SPLINE
SPL {X  -141.034, Y  +747.040, Z    +0.000, E1  +398.619, E3 -227248.265}
SPL {X  -152.334, Y  +720.400, Z    +0.000, E1  +389.143, E3 -227267.719}
SPL {X  -157.190, Y  +701.303, Z    +0.000, E1  +380.164, E3 -227274.880}
SPL {X  -159.117, Y  +688.191, Z    +0.000, E1  +372.748, E3 -227277.912}
SPL {X  -159.875, Y  +677.561, Z    +0.000, E1  +366.083, E3 -227279.302}
SPL {X  -159.990, Y  +669.975, Z    +0.000, E1  +360.595, E3 -227279.733}
SPL {X  -159.990, Y  +666.850, Z    +0.000, E1  +357.321, E3 -227279.833}
SPL {X  -159.990, Y  +662.495, Z    +0.000, E1  +351.318, E3 -227280.128}
SPL {X  -159.990, Y  +657.714, Z    +0.000, E1  +344.114, E3 -227280.689}
SPL {X  -159.990, Y  +651.822, Z    +0.000, E1  +335.261, E3 -227281.657}
SPL {X  -159.990, Y  +641.369, Z    +0.000, E1  +322.665, E3 -227284.495}
SPL {X  -159.990, Y  +598.251, Z    +0.000, E1  +304.104, E3 -227308.266}
SPL {X  -159.990, Y  +514.954, Z    +0.000, E1  +299.688, E3 -227382.062}
SPL {X  -159.990, Y  +505.641, Z    +0.000, E1  +299.707, E3 -227393.371}
SPL {X  -159.990, Y  +498.210, Z    +0.000, E1  +299.707, E3 -227402.364}
SPL {X  -159.990, Y  +488.988, Z    +0.000, E1  +299.693, E3 -227413.501}
SPL {X  -159.990, Y  +478.987, Z    +0.000, E1  +299.694, E3 -227425.604}
SPL {X  -159.990, Y  +468.796, Z    +0.000, E1  +299.698, E3 -227437.948}
SPL {X  -159.990, Y  +460.399, Z    +0.000, E1  +299.707, E3 -227448.124}
SPL {X  -159.990, Y  +453.289, Z    +0.000, E1  +299.707, E3 -227456.730}
SPL {X  -159.990, Y  +443.890, Z    +0.000, E1  +299.691, E3 -227468.083}
SPL {X  -159.990, Y  +437.910, Z    +0.000, E1  +300.175, E3 -227478.554}
ENDSPLINE

SPLINE
SPL {X  -159.990, Y  +447.165, Z    +0.000, E1  +303.287, E3 -227487.109}
ENDSPLINE

SPLINE
SPL {X  -159.990, Y  +436.354, Z    +0.000, E1  +302.683, E3 -227498.121}
SPL {X  -159.990, Y  +425.140, Z    +0.000, E1  +301.982, E3 -227508.556}
SPL {X  -159.990, Y  +412.625, Z    +0.000, E1  +301.150, E3 -227519.392}
SPL {X  -159.990, Y  +398.951, Z    +0.000, E1  +300.353, E3 -227531.264}
SPL {X  -159.990, Y  +389.564, Z    +0.000, E1  +300.093, E3 -227541.078}
SPL {X  -159.985, Y  +381.230, Z    +0.000, E1  +300.090, E3 -227551.345}
SPL {X  -159.702, Y  +372.900, Z    +0.000, E1  +300.135, E3 -227561.882}
SPL {X  -159.030, Y  +365.001, Z    +0.000, E1  +300.230, E3 -227572.284}
SPL {X  -157.449, Y  +354.098, Z    +0.000, E1  +300.447, E3 -227587.284}
SPL {X  -155.503, Y  +344.875, Z    +0.000, E1  +300.798, E3 -227600.703}
SPL {X  -153.622, Y  +337.813, Z    +0.000, E1  +301.097, E3 -227611.296}
SPL {X  -150.877, Y  +329.275, Z    +0.000, E1  +301.527, E3 -227624.521}
SPL {X  -148.134, Y  +322.059, Z    +0.000, E1  +302.038, E3 -227636.159}
SPL {X  -145.832, Y  +316.699, Z    +0.000, E1  +302.442, E3 -227644.994}
SPL {X  -143.160, Y  +311.071, Z    +0.000, E1  +302.918, E3 -227654.439}
SPL {X  -140.427, Y  +305.839, Z    +0.000, E1  +303.430, E3 -227663.400}
SPL {X  -137.611, Y  +300.891, Z    +0.000, E1  +303.950, E3 -227671.976}
SPL {X  -121.335, Y  +278.219, Z    +0.000, E1  +311.699, E3 -227770.322}
ENDSPLINE

SPLINE
SPL {X  -146.770, Y  +318.818, Z    +0.000, E1  +325.496, E3 -227870.156}
SPL {X  -156.430, Y  +348.936, Z    +0.000, E1  +338.153, E3 -227886.887}
SPL {X  -159.088, Y  +365.539, Z    +0.000, E1  +347.196, E3 -227891.298}
SPL {X  -159.820, Y  +375.127, Z    +0.000, E1  +353.170, E3 -227892.722}
SPL {X  -159.990, Y  +382.134, Z    +0.000, E1  +357.935, E3 -227893.240}
SPL {X  -159.990, Y  +385.595, Z    +0.000, E1  +360.838, E3 -227893.355}
SPL {X  -159.990, Y  +390.176, Z    +0.000, E1  +366.367, E3 -227893.624}
SPL {X  -159.990, Y  +395.747, Z    +0.000, E1  +374.484, E3 -227894.250}
SPL {X  -159.990, Y  +404.190, Z    +0.000, E1  +386.444, E3 -227895.932}
SPL {X  -159.990, Y  +418.143, Z    +0.000, E1  +401.167, E3 -227900.525}
SPL {X  -159.990, Y  +460.468, Z    +0.000, E1  +416.751, E3 -227923.207}
SPL {X  -159.990, Y  +537.348, Z    +0.000, E1  +420.157, E3 -227993.218}
SPL {X  -159.990, Y  +545.972, Z    +0.000, E1  +420.143, E3 -228003.752}
SPL {X  -159.990, Y  +557.131, Z    +0.000, E1  +420.184, E3 -228017.266}
SPL {X  -159.990, Y  +569.073, Z    +0.000, E1  +420.153, E3 -228031.861}
SPL {X  -159.990, Y  +577.562, Z    +0.000, E1  +420.146, E3 -228042.201}
SPL {X  -159.990, Y  +585.415, Z    +0.000, E1  +420.147, E3 -228051.767}
SPL {X  -159.990, Y  +594.125, Z    +0.000, E1  +420.153, E3 -228062.353}
SPL {X  -159.990, Y  +602.716, Z    +0.000, E1  +420.150, E3 -228072.816}
SPL {X  -159.990, Y  +612.205, Z    +0.000, E1  +420.159, E3 -228084.352}
SPL {X  -159.990, Y  +620.604, Z    +0.000, E1  +420.153, E3 -228094.568}
SPL {X  -159.990, Y  +632.106, Z    +0.000, E1  +420.183, E3 -228108.544}
SPL {X  -159.990, Y  +643.341, Z    +0.000, E1  +420.148, E3 -228122.288}
SPL {X  -159.990, Y  +652.098, Z    +0.000, E1  +420.153, E3 -228132.933}
SPL {X  -159.990, Y  +661.466, Z    +0.000, E1  +420.154, E3 -228144.345}
SPL {X  -159.990, Y  +670.781, Z    +0.000, E1  +420.150, E3 -228155.692}
SPL {X  -159.839, Y  +678.445, Z    +0.000, E1  +420.123, E3 -228165.172}
SPL {X  -159.339, Y  +685.922, Z    +0.000, E1  +420.057, E3 -228174.774}
SPL {X  -158.381, Y  +694.132, Z    +0.000, E1  +419.909, E3 -228185.771}
SPL {X  -157.192, Y  +701.291, Z    +0.000, E1  +419.715, E3 -228195.742}
SPL {X  -155.426, Y  +709.440, Z    +0.000, E1  +419.459, E3 -228207.440}
SPL {X  -153.239, Y  +717.485, Z    +0.000, E1  +419.087, E3 -228219.485}
SPL {X  -151.467, Y  +723.022, Z    +0.000, E1  +418.780, E3 -228228.037}
SPL {X  -148.791, Y  +730.306, Z    +0.000, E1  +418.370, E3 -228239.502}
SPL {X  -145.943, Y  +737.055, Z    +0.000, E1  +417.829, E3 -228250.555}
SPL {X  -143.898, Y  +741.430, Z    +0.000, E1  +417.467, E3 -228257.825}
SPL {X  -141.624, Y  +745.927, Z    +0.000, E1  +417.045, E3 -228265.420}
SPL {X  -139.581, Y  +749.692, Z    +0.000, E1  +416.662, E3 -228271.866}
SPL {X  -137.120, Y  +753.931, Z    +0.000, E1  +416.213, E3 -228279.164}
SPL {X  -120.054, Y  +777.254, Z    +0.000, E1  +409.463, E3 -228365.910}
ENDSPLINE

SPLINE
SPL {X  -141.034, Y  +747.040, Z    +0.000, E1  +398.619, E3 -228474.072}
SPL {X  -152.334, Y  +720.400, Z    +0.000, E1  +389.143, E3 -228493.526}
SPL {X  -157.190, Y  +701.303, Z    +0.000, E1  +380.164, E3 -228500.687}
SPL {X  -159.117, Y  +688.191, Z    +0.000, E1  +372.748, E3 -228503.719}
SPL {X  -159.875, Y  +677.561, Z    +0.000, E1  +366.083, E3 -228505.108}
SPL {X  -159.990, Y  +671.043, Z    +0.000, E1  +361.371, E3 -228505.512}
SPL {X  -159.990, Y  +668.657, Z    +0.000, E1  +359.332, E3 -228505.573}
SPL {X  -159.990, Y  +665.812, Z    +0.000, E1  +355.875, E3 -228505.684}
SPL {X  -159.990, Y  +662.495, Z    +0.000, E1  +351.318, E3 -228505.934}
SPL {X  -159.990, Y  +657.714, Z    +0.000, E1  +344.114, E3 -228506.495}
SPL {X  -159.990, Y  +651.822, Z    +0.000, E1  +335.261, E3 -228507.463}
SPL {X  -159.990, Y  +641.369, Z    +0.000, E1  +322.665, E3 -228510.301}
SPL {X  -159.990, Y  +598.251, Z    +0.000, E1  +304.104, E3 -228534.073}
SPL {X  -159.990, Y  +514.954, Z    +0.000, E1  +299.688, E3 -228607.868}
SPL {X  -159.990, Y  +505.641, Z    +0.000, E1  +299.707, E3 -228619.177}
SPL {X  -159.990, Y  +498.210, Z    +0.000, E1  +299.707, E3 -228628.171}
SPL {X  -159.990, Y  +488.988, Z    +0.000, E1  +299.693, E3 -228639.308}
SPL {X  -159.990, Y  +478.987, Z    +0.000, E1  +299.694, E3 -228651.410}
SPL {X  -159.990, Y  +468.796, Z    +0.000, E1  +299.698, E3 -228663.754}
SPL {X  -159.990, Y  +456.606, Z    +0.000, E1  +299.670, E3 -228678.460}
SPL {X  -159.990, Y  +443.890, Z    +0.000, E1  +299.691, E3 -228693.890}
SPL {X  -159.990, Y  +437.910, Z    +0.000, E1  +300.175, E3 -228704.361}
ENDSPLINE

SPLINE
SPL {X  -159.990, Y  +447.165, Z    +0.000, E1  +303.287, E3 -228712.916}
ENDSPLINE

SPLINE
SPL {X  -159.990, Y  +436.354, Z    +0.000, E1  +302.683, E3 -228723.927}
SPL {X  -159.990, Y  +425.140, Z    +0.000, E1  +301.982, E3 -228734.363}
SPL {X  -159.990, Y  +412.625, Z    +0.000, E1  +301.150, E3 -228745.199}
SPL {X  -159.990, Y  +398.951, Z    +0.000, E1  +300.353, E3 -228757.070}
SPL {X  -159.990, Y  +389.564, Z    +0.000, E1  +300.093, E3 -228766.884}
SPL {X  -159.985, Y  +381.230, Z    +0.000, E1  +300.090, E3 -228777.151}
SPL {X  -159.702, Y  +372.900, Z    +0.000, E1  +300.135, E3 -228787.688}
SPL {X  -159.030, Y  +365.001, Z    +0.000, E1  +300.230, E3 -228798.091}
SPL {X  -157.449, Y  +354.098, Z    +0.000, E1  +300.447, E3 -228813.090}
SPL {X  -155.503, Y  +344.875, Z    +0.000, E1  +300.798, E3 -228826.509}
SPL {X  -153.622, Y  +337.813, Z    +0.000, E1  +301.097, E3 -228837.102}
SPL {X  -151.786, Y  +331.925, Z    +0.000, E1  +301.419, E3 -228846.223}
SPL {X  -150.141, Y  +327.233, Z    +0.000, E1  +301.695, E3 -228853.632}
SPL {X  -148.134, Y  +322.059, Z    +0.000, E1  +302.038, E3 -228861.966}
SPL {X  -145.832, Y  +316.699, Z    +0.000, E1  +302.442, E3 -228870.800}
SPL {X  -143.160, Y  +311.071, Z    +0.000, E1  +302.918, E3 -228880.245}
SPL {X  -140.427, Y  +305.839, Z    +0.000, E1  +303.430, E3 -228889.207}
SPL {X  -137.611, Y  +300.891, Z    +0.000, E1  +303.950, E3 -228897.783}
SPL {X  -121.335, Y  +278.219, Z    +0.000, E1  +311.699, E3 -228996.129}
ENDSPLINE

SPLINE
SPL {X  -146.770, Y  +318.818, Z    +0.000, E1  +325.496, E3 -229095.963}
SPL {X  -156.430, Y  +348.936, Z    +0.000, E1  +338.153, E3 -229112.694}
SPL {X  -159.088, Y  +365.539, Z    +0.000, E1  +347.196, E3 -229117.105}
SPL {X  -159.921, Y  +377.798, Z    +0.000, E1  +354.872, E3 -229118.765}
SPL {X  -159.990, Y  +384.169, Z    +0.000, E1  +359.534, E3 -229119.120}
SPL {X  -159.990, Y  +386.366, Z    +0.000, E1  +361.774, E3 -229119.185}
SPL {X  -159.990, Y  +390.176, Z    +0.000, E1  +366.367, E3 -229119.431}
SPL {X  -159.990, Y  +395.747, Z    +0.000, E1  +374.484, E3 -229120.056}
SPL {X  -159.990, Y  +402.387, Z    +0.000, E1  +384.140, E3 -229121.289}
SPL {X  -159.990, Y  +414.244, Z    +0.000, E1  +397.704, E3 -229124.921}
SPL {X  -159.990, Y  +460.468, Z    +0.000, E1  +416.751, E3 -229149.013}
SPL {X  -159.990, Y  +537.348, Z    +0.000, E1  +420.157, E3 -229219.025}
SPL {X  -159.990, Y  +549.907, Z    +0.000, E1  +420.183, E3 -229234.282}
SPL {X  -159.990, Y  +560.677, Z    +0.000, E1  +420.145, E3 -229247.453}
SPL {X  -159.990, Y  +569.073, Z    +0.000, E1  +420.153, E3 -229257.668}
SPL {X  -159.990, Y  +577.562, Z    +0.000, E1  +420.146, E3 -229268.008}
SPL {X  -159.990, Y  +585.415, Z    +0.000, E1  +420.147, E3 -229277.573}
SPL {X  -159.990, Y  +594.125, Z    +0.000, E1  +420.153, E3 -229288.159}
SPL {X  -159.990, Y  +602.716, Z    +0.000, E1  +420.150, E3 -229298.622}
SPL {X  -159.990, Y  +612.205, Z    +0.000, E1  +420.159, E3 -229310.159}
SPL {X  -159.990, Y  +624.752, Z    +0.000, E1  +420.194, E3 -229325.367}
SPL {X  -159.990, Y  +640.062, Z    +0.000, E1  +420.188, E3 -229344.030}
SPL {X  -159.990, Y  +652.098, Z    +0.000, E1  +420.153, E3 -229358.740}
SPL {X  -159.990, Y  +661.466, Z    +0.000, E1  +420.154, E3 -229370.151}
SPL {X  -159.963, Y  +674.441, Z    +0.000, E1  +420.189, E3 -229385.902}
SPL {X  -159.339, Y  +685.922, Z    +0.000, E1  +420.057, E3 -229400.581}
SPL {X  -158.381, Y  +694.132, Z    +0.000, E1  +419.909, E3 -229411.578}
SPL {X  -156.712, Y  +703.719, Z    +0.000, E1  +419.674, E3 -229424.943}
SPL {X  -154.922, Y  +711.450, Z    +0.000, E1  +419.348, E3 -229436.259}
SPL {X  -153.239, Y  +717.485, Z    +0.000, E1  +419.087, E3 -229445.291}
SPL {X  -150.608, Y  +725.483, Z    +0.000, E1  +418.677, E3 -229457.637}
SPL {X  -148.008, Y  +732.249, Z    +0.000, E1  +418.192, E3 -229468.503}
SPL {X  -145.943, Y  +737.055, Z    +0.000, E1  +417.829, E3 -229476.362}
SPL {X  -143.898, Y  +741.430, Z    +0.000, E1  +417.467, E3 -229483.631}
SPL {X  -141.624, Y  +745.927, Z    +0.000, E1  +417.045, E3 -229491.226}
SPL {X  -139.581, Y  +749.692, Z    +0.000, E1  +416.662, E3 -229497.673}
SPL {X  -137.120, Y  +753.931, Z    +0.000, E1  +416.213, E3 -229504.970}
SPL {X  -120.054, Y  +777.254, Z    +0.000, E1  +409.463, E3 -229591.716}
ENDSPLINE

SPLINE
SPL {X  -141.034, Y  +747.040, Z    +0.000, E1  +398.619, E3 -229699.878}
SPL {X  -152.334, Y  +720.400, Z    +0.000, E1  +389.143, E3 -229719.332}
SPL {X  -157.190, Y  +701.303, Z    +0.000, E1  +380.164, E3 -229726.493}
SPL {X  -159.460, Y  +684.516, Z    +0.000, E1  +370.556, E3 -229730.089}
SPL {X  -159.938, Y  +675.597, Z    +0.000, E1  +364.669, E3 -229731.095}
SPL {X  -159.990, Y  +671.043, Z    +0.000, E1  +361.371, E3 -229731.319}
SPL {X  -159.990, Y  +668.657, Z    +0.000, E1  +359.332, E3 -229731.379}
SPL {X  -159.990, Y  +665.812, Z    +0.000, E1  +355.875, E3 -229731.491}
SPL {X  -159.990, Y  +662.495, Z    +0.000, E1  +351.318, E3 -229731.740}
SPL {X  -159.990, Y  +657.714, Z    +0.000, E1  +344.114, E3 -229732.302}
SPL {X  -159.990, Y  +651.822, Z    +0.000, E1  +335.261, E3 -229733.270}
SPL {X  -159.990, Y  +641.369, Z    +0.000, E1  +322.665, E3 -229736.108}
SPL {X  -159.990, Y  +598.251, Z    +0.000, E1  +304.104, E3 -229759.879}
SPL {X  -159.990, Y  +514.954, Z    +0.000, E1  +299.688, E3 -229833.675}
SPL {X  -159.990, Y  +505.641, Z    +0.000, E1  +299.707, E3 -229844.984}
SPL {X  -159.990, Y  +498.210, Z    +0.000, E1  +299.707, E3 -229853.977}
SPL {X  -159.990, Y  +488.988, Z    +0.000, E1  +299.693, E3 -229865.114}
SPL {X  -159.990, Y  +478.987, Z    +0.000, E1  +299.694, E3 -229877.217}
SPL {X  -159.990, Y  +468.796, Z    +0.000, E1  +299.698, E3 -229889.561}
SPL {X  -159.990, Y  +456.606, Z    +0.000, E1  +299.670, E3 -229904.266}
SPL {X  -159.990, Y  +443.890, Z    +0.000, E1  +299.691, E3 -229919.696}
SPL {X  -159.990, Y  +437.910, Z    +0.000, E1  +300.175, E3 -229930.167}
ENDSPLINE

SPLINE
SPL {X  -159.990, Y  +447.165, Z    +0.000, E1  +303.287, E3 -229938.722}
ENDSPLINE

SPLINE
SPL {X  -159.990, Y  +436.354, Z    +0.000, E1  +302.683, E3 -229949.734}
SPL {X  -159.990, Y  +425.140, Z    +0.000, E1  +301.982, E3 -229960.169}
SPL {X  -159.990, Y  +412.625, Z    +0.000, E1  +301.150, E3 -229971.005}
SPL {X  -159.990, Y  +398.951, Z    +0.000, E1  +300.353, E3 -229982.877}
SPL {X  -159.990, Y  +389.564, Z    +0.000, E1  +300.093, E3 -229992.690}
SPL {X  -159.985, Y  +381.230, Z    +0.000, E1  +300.090, E3 -230002.957}
SPL {X  -159.702, Y  +372.900, Z    +0.000, E1  +300.135, E3 -230013.494}
SPL {X  -159.030, Y  +365.001, Z    +0.000, E1  +300.230, E3 -230023.897}
SPL {X  -158.029, Y  +357.528, Z    +0.000, E1  +300.403, E3 -230034.153}
SPL {X  -156.953, Y  +351.476, Z    +0.000, E1  +300.570, E3 -230042.706}
SPL {X  -155.503, Y  +344.875, Z    +0.000, E1  +300.798, E3 -230052.316}
SPL {X  -153.622, Y  +337.813, Z    +0.000, E1  +301.097, E3 -230062.909}
SPL {X  -150.877, Y  +329.275, Z    +0.000, E1  +301.527, E3 -230076.134}
SPL {X  -148.134, Y  +322.059, Z    +0.000, E1  +302.038, E3 -230087.772}
SPL {X  -145.832, Y  +316.699, Z    +0.000, E1  +302.442, E3 -230096.607}
SPL {X  -143.160, Y  +311.071, Z    +0.000, E1  +302.918, E3 -230106.052}
SPL {X  -139.570, Y  +304.288, Z    +0.000, E1  +303.552, E3 -230117.648}
SPL {X  -136.734, Y  +299.430, Z    +0.000, E1  +304.147, E3 -230126.186}
SPL {X  -121.335, Y  +278.219, Z    +0.000, E1  +311.699, E3 -230221.935}
ENDSPLINE

SPLINE
SPL {X  -146.770, Y  +318.818, Z    +0.000, E1  +325.496, E3 -230321.769}
SPL {X  -156.430, Y  +348.936, Z    +0.000, E1  +338.153, E3 -230338.500}
SPL {X  -159.088, Y  +365.539, Z    +0.000, E1  +347.196, E3 -230342.911}
SPL {X  -159.921, Y  +377.798, Z    +0.000, E1  +354.872, E3 -230344.571}
SPL {X  -159.990, Y  +383.148, Z    +0.000, E1  +358.786, E3 -230344.899}
SPL {X  -159.990, Y  +384.761, Z    +0.000, E1  +360.138, E3 -230344.943}
SPL {X  -159.990, Y  +387.385, Z    +0.000, E1  +362.811, E3 -230345.045}
SPL {X  -159.990, Y  +391.439, Z    +0.000, E1  +368.259, E3 -230345.342}
SPL {X  -159.990, Y  +395.747, Z    +0.000, E1  +374.484, E3 -230345.863}
SPL {X  -159.990, Y  +402.387, Z    +0.000, E1  +384.140, E3 -230347.095}
SPL {X  -159.990, Y  +414.244, Z    +0.000, E1  +397.704, E3 -230350.728}
SPL {X  -159.990, Y  +460.468, Z    +0.000, E1  +416.751, E3 -230374.820}
SPL {X  -159.990, Y  +537.348, Z    +0.000, E1  +420.157, E3 -230444.831}
SPL {X  -159.990, Y  +549.907, Z    +0.000, E1  +420.183, E3 -230460.089}
SPL {X  -159.990, Y  +560.677, Z    +0.000, E1  +420.145, E3 -230473.260}
SPL {X  -159.990, Y  +569.073, Z    +0.000, E1  +420.153, E3 -230483.474}
SPL {X  -159.990, Y  +581.828, Z    +0.000, E1  +420.191, E3 -230498.933}
SPL {X  -159.990, Y  +594.125, Z    +0.000, E1  +420.153, E3 -230513.966}
SPL {X  -159.990, Y  +602.716, Z    +0.000, E1  +420.150, E3 -230524.429}
SPL {X  -159.990, Y  +612.205, Z    +0.000, E1  +420.159, E3 -230535.965}
SPL {X  -159.990, Y  +620.604, Z    +0.000, E1  +420.153, E3 -230546.181}
SPL {X  -159.990, Y  +632.106, Z    +0.000, E1  +420.183, E3 -230560.157}
SPL {X  -159.990, Y  +643.341, Z    +0.000, E1  +420.148, E3 -230573.901}
SPL {X  -159.990, Y  +652.098, Z    +0.000, E1  +420.153, E3 -230584.546}
SPL {X  -159.990, Y  +661.466, Z    +0.000, E1  +420.154, E3 -230595.958}
SPL {X  -159.990, Y  +670.781, Z    +0.000, E1  +420.150, E3 -230607.305}
SPL {X  -159.839, Y  +678.445, Z    +0.000, E1  +420.123, E3 -230616.785}
SPL {X  -159.339, Y  +685.922, Z    +0.000, E1  +420.057, E3 -230626.387}
SPL {X  -158.381, Y  +694.132, Z    +0.000, E1  +419.909, E3 -230637.384}
SPL {X  -157.192, Y  +701.291, Z    +0.000, E1  +419.715, E3 -230647.355}
SPL {X  -155.426, Y  +709.440, Z    +0.000, E1  +419.459, E3 -230659.053}
SPL {X  -153.239, Y  +717.485, Z    +0.000, E1  +419.087, E3 -230671.098}
SPL {X  -151.467, Y  +723.022, Z    +0.000, E1  +418.780, E3 -230679.650}
SPL {X  -148.791, Y  +730.306, Z    +0.000, E1  +418.370, E3 -230691.115}
SPL {X  -145.943, Y  +737.055, Z    +0.000, E1  +417.829, E3 -230702.168}
SPL {X  -143.898, Y  +741.430, Z    +0.000, E1  +417.467, E3 -230709.437}
SPL {X  -140.579, Y  +747.882, Z    +0.000, E1  +416.895, E3 -230720.316}
SPL {X  -137.120, Y  +753.931, Z    +0.000, E1  +416.213, E3 -230730.777}
SPL {X  -120.054, Y  +777.254, Z    +0.000, E1  +409.463, E3 -230817.523}
ENDSPLINE

SPLINE
SPL {X  -141.034, Y  +747.040, Z    +0.000, E1  +398.619, E3 -230925.685}
SPL {X  -152.334, Y  +720.400, Z    +0.000, E1  +389.143, E3 -230945.139}
SPL {X  -157.190, Y  +701.303, Z    +0.000, E1  +380.164, E3 -230952.299}
SPL {X  -159.460, Y  +684.516, Z    +0.000, E1  +370.556, E3 -230955.895}
SPL {X  -159.938, Y  +675.597, Z    +0.000, E1  +364.669, E3 -230956.902}
SPL {X  -159.990, Y  +671.043, Z    +0.000, E1  +361.371, E3 -230957.125}
SPL {X  -159.990, Y  +668.657, Z    +0.000, E1  +359.332, E3 -230957.186}
SPL {X  -159.990, Y  +665.812, Z    +0.000, E1  +355.875, E3 -230957.297}
SPL {X  -159.990, Y  +662.495, Z    +0.000, E1  +351.318, E3 -230957.547}
SPL {X  -159.990, Y  +657.714, Z    +0.000, E1  +344.114, E3 -230958.108}
SPL {X  -159.990, Y  +651.822, Z    +0.000, E1  +335.261, E3 -230959.076}
SPL {X  -159.990, Y  +641.369, Z    +0.000, E1  +322.665, E3 -230961.914}
SPL {X  -159.990, Y  +598.251, Z    +0.000, E1  +304.104, E3 -230985.686}
SPL {X  -159.990, Y  +514.954, Z    +0.000, E1  +299.688, E3 -231059.481}
SPL {X  -159.990, Y  +505.641, Z    +0.000, E1  +299.707, E3 -231070.790}
SPL {X  -159.990, Y  +498.210, Z    +0.000, E1  +299.707, E3 -231079.784}
SPL {X  -159.990, Y  +488.988, Z    +0.000, E1  +299.693, E3 -231090.921}
SPL {X  -159.990, Y  +478.987, Z    +0.000, E1  +299.694, E3 -231103.023}
SPL {X  -159.990, Y  +468.796, Z    +0.000, E1  +299.698, E3 -231115.367}
SPL {X  -159.990, Y  +460.399, Z    +0.000, E1  +299.707, E3 -231125.544}
SPL {X  -159.990, Y  +453.289, Z    +0.000, E1  +299.707, E3 -231134.149}
SPL {X  -159.990, Y  +443.890, Z    +0.000, E1  +299.691, E3 -231145.503}
SPL {X  -159.990, Y  +437.910, Z    +0.000, E1  +300.175, E3 -231155.974}
ENDSPLINE

SPLINE
SPL {X  -159.990, Y  +447.165, Z    +0.000, E1  +303.287, E3 -231164.529}
ENDSPLINE

SPLINE
SPL {X  -159.990, Y  +436.354, Z    +0.000, E1  +302.683, E3 -231175.540}
SPL {X  -159.990, Y  +425.140, Z    +0.000, E1  +301.982, E3 -231185.976}
SPL {X  -159.990, Y  +412.625, Z    +0.000, E1  +301.150, E3 -231196.812}
SPL {X  -159.990, Y  +398.951, Z    +0.000, E1  +300.353, E3 -231208.683}
SPL {X  -159.990, Y  +389.564, Z    +0.000, E1  +300.093, E3 -231218.497}
SPL {X  -159.985, Y  +381.230, Z    +0.000, E1  +300.090, E3 -231228.764}
SPL {X  -159.702, Y  +372.900, Z    +0.000, E1  +300.135, E3 -231239.301}
SPL {X  -159.030, Y  +365.001, Z    +0.000, E1  +300.230, E3 -231249.704}
SPL {X  -158.029, Y  +357.528, Z    +0.000, E1  +300.403, E3 -231259.959}
SPL {X  -156.953, Y  +351.476, Z    +0.000, E1  +300.570, E3 -231268.512}
SPL {X  -155.503, Y  +344.875, Z    +0.000, E1  +300.798, E3 -231278.122}
SPL {X  -153.622, Y  +337.813, Z    +0.000, E1  +301.097, E3 -231288.715}
SPL {X  -150.877, Y  +329.275, Z    +0.000, E1  +301.527, E3 -231301.940}
SPL {X  -148.134, Y  +322.059, Z    +0.000, E1  +302.038, E3 -231313.579}
SPL {X  -145.832, Y  +316.699, Z    +0.000, E1  +302.442, E3 -231322.413}
SPL {X  -143.160, Y  +311.071, Z    +0.000, E1  +302.918, E3 -231331.858}
SPL {X  -140.427, Y  +305.839, Z    +0.000, E1  +303.430, E3 -231340.819}
SPL {X  -137.611, Y  +300.891, Z    +0.000, E1  +303.950, E3 -231349.396}
SPL {X  -121.335, Y  +278.219, Z    +0.000, E1  +311.699, E3 -231447.742}
ENDSPLINE

SPLINE
SPL {X  -146.770, Y  +318.818, Z    +0.000, E1  +325.496, E3 -231547.575}
SPL {X  -156.430, Y  +348.936, Z    +0.000, E1  +338.153, E3 -231564.307}
SPL {X  -159.088, Y  +365.539, Z    +0.000, E1  +347.196, E3 -231568.718}
SPL {X  -159.921, Y  +377.798, Z    +0.000, E1  +354.872, E3 -231570.378}
SPL {X  -159.990, Y  +384.169, Z    +0.000, E1  +359.534, E3 -231570.733}
SPL {X  -159.990, Y  +387.385, Z    +0.000, E1  +362.811, E3 -231570.852}
SPL {X  -159.990, Y  +391.439, Z    +0.000, E1  +368.259, E3 -231571.148}
SPL {X  -159.990, Y  +395.747, Z    +0.000, E1  +374.484, E3 -231571.669}
SPL {X  -159.990, Y  +402.387, Z    +0.000, E1  +384.140, E3 -231572.902}
SPL {X  -159.990, Y  +414.244, Z    +0.000, E1  +397.704, E3 -231576.534}
SPL {X  -159.990, Y  +460.468, Z    +0.000, E1  +416.751, E3 -231600.626}
SPL {X  -159.990, Y  +537.348, Z    +0.000, E1  +420.157, E3 -231670.638}
SPL {X  -159.990, Y  +545.972, Z    +0.000, E1  +420.143, E3 -231681.172}
SPL {X  -159.990, Y  +557.131, Z    +0.000, E1  +420.184, E3 -231694.686}
SPL {X  -159.990, Y  +569.073, Z    +0.000, E1  +420.153, E3 -231709.281}
SPL {X  -159.990, Y  +577.562, Z    +0.000, E1  +420.146, E3 -231719.621}
SPL {X  -159.990, Y  +585.415, Z    +0.000, E1  +420.147, E3 -231729.186}
SPL {X  -159.990, Y  +594.125, Z    +0.000, E1  +420.153, E3 -231739.772}
SPL {X  -159.990, Y  +602.716, Z    +0.000, E1  +420.150, E3 -231750.235}
SPL {X  -159.990, Y  +612.205, Z    +0.000, E1  +420.159, E3 -231761.772}
SPL {X  -159.990, Y  +624.752, Z    +0.000, E1  +420.194, E3 -231776.980}
SPL {X  -159.990, Y  +640.062, Z    +0.000, E1  +420.188, E3 -231795.643}
SPL {X  -159.990, Y  +652.098, Z    +0.000, E1  +420.153, E3 -231810.353}
SPL {X  -159.990, Y  +661.466, Z    +0.000, E1  +420.154, E3 -231821.764}
SPL {X  -159.963, Y  +674.441, Z    +0.000, E1  +420.189, E3 -231837.515}
SPL {X  -159.339, Y  +685.922, Z    +0.000, E1  +420.057, E3 -231852.194}
SPL {X  -158.381, Y  +694.132, Z    +0.000, E1  +419.909, E3 -231863.191}
SPL {X  -156.712, Y  +703.719, Z    +0.000, E1  +419.674, E3 -231876.556}
SPL {X  -154.922, Y  +711.450, Z    +0.000, E1  +419.348, E3 -231887.872}
SPL {X  -153.239, Y  +717.485, Z    +0.000, E1  +419.087, E3 -231896.904}
SPL {X  -150.608, Y  +725.483, Z    +0.000, E1  +418.677, E3 -231909.249}
SPL {X  -148.008, Y  +732.249, Z    +0.000, E1  +418.192, E3 -231920.116}
SPL {X  -145.943, Y  +737.055, Z    +0.000, E1  +417.829, E3 -231927.975}
SPL {X  -143.898, Y  +741.430, Z    +0.000, E1  +417.467, E3 -231935.244}
SPL {X  -141.624, Y  +745.927, Z    +0.000, E1  +417.045, E3 -231942.839}
SPL {X  -139.581, Y  +749.692, Z    +0.000, E1  +416.662, E3 -231949.286}
SPL {X  -137.120, Y  +753.931, Z    +0.000, E1  +416.213, E3 -231956.583}
SPL {X  -120.054, Y  +777.254, Z    +0.000, E1  +409.463, E3 -232043.329}
ENDSPLINE

SPLINE
SPL {X  -141.034, Y  +747.040, Z    +0.000, E1  +398.619, E3 -232151.491}
SPL {X  -152.334, Y  +720.400, Z    +0.000, E1  +389.143, E3 -232170.945}
SPL {X  -157.190, Y  +701.303, Z    +0.000, E1  +380.164, E3 -232178.106}
SPL {X  -159.460, Y  +684.516, Z    +0.000, E1  +370.556, E3 -232181.701}
SPL {X  -159.938, Y  +675.597, Z    +0.000, E1  +364.669, E3 -232182.708}
SPL {X  -159.990, Y  +671.043, Z    +0.000, E1  +361.371, E3 -232182.932}
SPL {X  -159.990, Y  +668.657, Z    +0.000, E1  +359.332, E3 -232182.992}
SPL {X  -159.990, Y  +665.812, Z    +0.000, E1  +355.875, E3 -232183.104}
SPL {X  -159.990, Y  +662.495, Z    +0.000, E1  +351.318, E3 -232183.353}
SPL {X  -159.990, Y  +657.714, Z    +0.000, E1  +344.114, E3 -232183.914}
SPL {X  -159.990, Y  +651.822, Z    +0.000, E1  +335.261, E3 -232184.883}
SPL {X  -159.990, Y  +641.369, Z    +0.000, E1  +322.665, E3 -232187.721}
SPL {X  -159.990, Y  +598.251, Z    +0.000, E1  +304.104, E3 -232211.492}
SPL {X  -159.990, Y  +514.954, Z    +0.000, E1  +299.688, E3 -232285.288}
SPL {X  -159.990, Y  +505.641, Z    +0.000, E1  +299.707, E3 -232296.597}
SPL {X  -159.990, Y  +498.210, Z    +0.000, E1  +299.707, E3 -232305.590}
SPL {X  -159.990, Y  +488.988, Z    +0.000, E1  +299.693, E3 -232316.727}
SPL {X  -159.990, Y  +478.987, Z    +0.000, E1  +299.694, E3 -232328.830}
SPL {X  -159.990, Y  +468.796, Z    +0.000, E1  +299.698, E3 -232341.173}
SPL {X  -159.990, Y  +456.606, Z    +0.000, E1  +299.670, E3 -232355.879}
SPL {X  -159.990, Y  +443.890, Z    +0.000, E1  +299.691, E3 -232371.309}
SPL {X  -159.990, Y  +437.910, Z    +0.000, E1  +300.175, E3 -232381.780}
ENDSPLINE

SPLINE
SPL {X  -159.990, Y  +447.165, Z    +0.000, E1  +303.287, E3 -232390.335}
ENDSPLINE

SPLINE
SPL {X  -159.990, Y  +436.354, Z    +0.000, E1  +302.683, E3 -232401.347}
SPL {X  -159.990, Y  +425.140, Z    +0.000, E1  +301.982, E3 -232411.782}
SPL {X  -159.990, Y  +412.625, Z    +0.000, E1  +301.150, E3 -232422.618}
SPL {X  -159.990, Y  +398.951, Z    +0.000, E1  +300.353, E3 -232434.489}
SPL {X  -159.990, Y  +389.564, Z    +0.000, E1  +300.093, E3 -232444.303}
SPL {X  -159.985, Y  +381.230, Z    +0.000, E1  +300.090, E3 -232454.570}
SPL {X  -159.702, Y  +372.900, Z    +0.000, E1  +300.135, E3 -232465.107}
SPL {X  -159.030, Y  +365.001, Z    +0.000, E1  +300.230, E3 -232475.510}
SPL {X  -158.029, Y  +357.528, Z    +0.000, E1  +300.403, E3 -232485.766}
SPL {X  -156.953, Y  +351.476, Z    +0.000, E1  +300.570, E3 -232494.319}
SPL {X  -155.503, Y  +344.875, Z    +0.000, E1  +300.798, E3 -232503.928}
SPL {X  -153.622, Y  +337.813, Z    +0.000, E1  +301.097, E3 -232514.522}
SPL {X  -150.877, Y  +329.275, Z    +0.000, E1  +301.527, E3 -232527.747}
SPL {X  -148.134, Y  +322.059, Z    +0.000, E1  +302.038, E3 -232539.385}
SPL {X  -145.832, Y  +316.699, Z    +0.000, E1  +302.442, E3 -232548.220}
SPL {X  -143.160, Y  +311.071, Z    +0.000, E1  +302.918, E3 -232557.665}
SPL {X  -139.570, Y  +304.288, Z    +0.000, E1  +303.552, E3 -232569.261}
SPL {X  -136.734, Y  +299.430, Z    +0.000, E1  +304.147, E3 -232577.799}
SPL {X  -121.335, Y  +278.219, Z    +0.000, E1  +311.699, E3 -232673.548}
ENDSPLINE

SPLINE
SPL {X  -146.770, Y  +318.818, Z    +0.000, E1  +325.496, E3 -232773.382}
SPL {X  -156.430, Y  +348.936, Z    +0.000, E1  +338.153, E3 -232790.113}
SPL {X  -159.088, Y  +365.539, Z    +0.000, E1  +347.196, E3 -232794.524}
SPL {X  -159.921, Y  +377.798, Z    +0.000, E1  +354.872, E3 -232796.184}
SPL {X  -159.990, Y  +383.148, Z    +0.000, E1  +358.786, E3 -232796.512}
SPL {X  -159.990, Y  +384.761, Z    +0.000, E1  +360.138, E3 -232796.556}
SPL {X  -159.990, Y  +387.385, Z    +0.000, E1  +362.811, E3 -232796.658}
SPL {X  -159.990, Y  +391.439, Z    +0.000, E1  +368.259, E3 -232796.955}
SPL {X  -159.990, Y  +395.747, Z    +0.000, E1  +374.484, E3 -232797.475}
SPL {X  -159.990, Y  +402.387, Z    +0.000, E1  +384.140, E3 -232798.708}
SPL {X  -159.990, Y  +414.244, Z    +0.000, E1  +397.704, E3 -232802.341}
SPL {X  -159.990, Y  +460.468, Z    +0.000, E1  +416.751, E3 -232826.433}
SPL {X  -159.990, Y  +537.348, Z    +0.000, E1  +420.157, E3 -232896.444}
SPL {X  -159.990, Y  +549.907, Z    +0.000, E1  +420.183, E3 -232911.702}
SPL {X  -159.990, Y  +560.677, Z    +0.000, E1  +420.145, E3 -232924.873}
SPL {X  -159.990, Y  +569.073, Z    +0.000, E1  +420.153, E3 -232935.087}
SPL {X  -159.990, Y  +581.828, Z    +0.000, E1  +420.191, E3 -232950.546}
SPL {X  -159.990, Y  +594.125, Z    +0.000, E1  +420.153, E3 -232965.579}
SPL {X  -159.990, Y  +602.716, Z    +0.000, E1  +420.150, E3 -232976.042}
SPL {X  -159.990, Y  +612.205, Z    +0.000, E1  +420.159, E3 -232987.578}
SPL {X  -159.990, Y  +620.604, Z    +0.000, E1  +420.153, E3 -232997.794}
SPL {X  -159.990, Y  +632.106, Z    +0.000, E1  +420.183, E3 -233011.770}
SPL {X  -159.990, Y  +643.341, Z    +0.000, E1  +420.148, E3 -233025.514}
SPL {X  -159.990, Y  +652.098, Z    +0.000, E1  +420.153, E3 -233036.159}
SPL {X  -159.990, Y  +661.466, Z    +0.000, E1  +420.154, E3 -233047.571}
SPL {X  -159.990, Y  +670.781, Z    +0.000, E1  +420.150, E3 -233058.918}
SPL {X  -159.839, Y  +678.445, Z    +0.000, E1  +420.123, E3 -233068.398}
SPL {X  -159.339, Y  +685.922, Z    +0.000, E1  +420.057, E3 -233078.000}
SPL {X  -158.381, Y  +694.132, Z    +0.000, E1  +419.909, E3 -233088.997}
SPL {X  -157.192, Y  +701.291, Z    +0.000, E1  +419.715, E3 -233098.968}
SPL {X  -155.426, Y  +709.440, Z    +0.000, E1  +419.459, E3 -233110.665}
SPL {X  -153.239, Y  +717.485, Z    +0.000, E1  +419.087, E3 -233122.711}
SPL {X  -151.467, Y  +723.022, Z    +0.000, E1  +418.780, E3 -233131.263}
SPL {X  -148.791, Y  +730.306, Z    +0.000, E1  +418.370, E3 -233142.728}
SPL {X  -145.943, Y  +737.055, Z    +0.000, E1  +417.829, E3 -233153.781}
SPL {X  -143.898, Y  +741.430, Z    +0.000, E1  +417.467, E3 -233161.050}
SPL {X  -140.579, Y  +747.882, Z    +0.000, E1  +416.895, E3 -233171.929}
SPL {X  -137.120, Y  +753.931, Z    +0.000, E1  +416.213, E3 -233182.390}
SPL {X  -120.054, Y  +777.254, Z    +0.000, E1  +409.463, E3 -233269.136}
ENDSPLINE

SPLINE
SPL {X  -141.034, Y  +747.040, Z    +0.000, E1  +398.619, E3 -233377.297}
SPL {X  -152.334, Y  +720.400, Z    +0.000, E1  +389.143, E3 -233396.752}
SPL {X  -157.190, Y  +701.303, Z    +0.000, E1  +380.164, E3 -233403.912}
SPL {X  -159.460, Y  +684.516, Z    +0.000, E1  +370.556, E3 -233407.508}
SPL {X  -159.938, Y  +675.597, Z    +0.000, E1  +364.669, E3 -233408.514}
SPL {X  -159.990, Y  +671.043, Z    +0.000, E1  +361.371, E3 -233408.738}
SPL {X  -159.990, Y  +668.657, Z    +0.000, E1  +359.332, E3 -233408.799}
SPL {X  -159.990, Y  +665.812, Z    +0.000, E1  +355.875, E3 -233408.910}
SPL {X  -159.990, Y  +662.495, Z    +0.000, E1  +351.318, E3 -233409.160}
SPL {X  -159.990, Y  +657.714, Z    +0.000, E1  +344.114, E3 -233409.721}
SPL {X  -159.990, Y  +651.822, Z    +0.000, E1  +335.261, E3 -233410.689}
SPL {X  -159.990, Y  +641.369, Z    +0.000, E1  +322.665, E3 -233413.527}
SPL {X  -159.990, Y  +598.251, Z    +0.000, E1  +304.104, E3 -233437.299}
SPL {X  -159.990, Y  +514.954, Z    +0.000, E1  +299.688, E3 -233511.094}
SPL {X  -159.990, Y  +505.641, Z    +0.000, E1  +299.707, E3 -233522.403}
SPL {X  -159.990, Y  +498.210, Z    +0.000, E1  +299.707, E3 -233531.397}
SPL {X  -159.990, Y  +488.988, Z    +0.000, E1  +299.693, E3 -233542.534}
SPL {X  -159.990, Y  +478.987, Z    +0.000, E1  +299.694, E3 -233554.636}
SPL {X  -159.990, Y  +468.796, Z    +0.000, E1  +299.698, E3 -233566.980}
SPL {X  -159.990, Y  +460.399, Z    +0.000, E1  +299.707, E3 -233577.157}
SPL {X  -159.990, Y  +453.289, Z    +0.000, E1  +299.707, E3 -233585.762}
SPL {X  -159.990, Y  +443.890, Z    +0.000, E1  +299.691, E3 -233597.116}
SPL {X  -159.990, Y  +437.910, Z    +0.000, E1  +300.175, E3 -233607.587}
ENDSPLINE

SPLINE
SPL {X  -159.990, Y  +447.165, Z    +0.000, E1  +303.287, E3 -233616.142}
ENDSPLINE

SPLINE
SPL {X  -159.990, Y  +436.354, Z    +0.000, E1  +302.683, E3 -233627.153}
SPL {X  -159.990, Y  +425.140, Z    +0.000, E1  +301.982, E3 -233637.589}
SPL {X  -159.990, Y  +412.625, Z    +0.000, E1  +301.150, E3 -233648.425}
SPL {X  -159.990, Y  +398.951, Z    +0.000, E1  +300.353, E3 -233660.296}
SPL {X  -159.990, Y  +389.564, Z    +0.000, E1  +300.093, E3 -233670.110}
SPL {X  -159.985, Y  +381.230, Z    +0.000, E1  +300.090, E3 -233680.377}
SPL {X  -159.702, Y  +372.900, Z    +0.000, E1  +300.135, E3 -233690.914}
SPL {X  -159.030, Y  +365.001, Z    +0.000, E1  +300.230, E3 -233701.317}
SPL {X  -158.029, Y  +357.528, Z    +0.000, E1  +300.403, E3 -233711.572}
SPL {X  -156.953, Y  +351.476, Z    +0.000, E1  +300.570, E3 -233720.125}
SPL {X  -155.503, Y  +344.875, Z    +0.000, E1  +300.798, E3 -233729.735}
SPL {X  -153.622, Y  +337.813, Z    +0.000, E1  +301.097, E3 -233740.328}
SPL {X  -150.877, Y  +329.275, Z    +0.000, E1  +301.527, E3 -233753.553}
SPL {X  -148.134, Y  +322.059, Z    +0.000, E1  +302.038, E3 -233765.192}
SPL {X  -145.832, Y  +316.699, Z    +0.000, E1  +302.442, E3 -233774.026}
SPL {X  -143.160, Y  +311.071, Z    +0.000, E1  +302.918, E3 -233783.471}
SPL {X  -140.427, Y  +305.839, Z    +0.000, E1  +303.430, E3 -233792.432}
SPL {X  -137.611, Y  +300.891, Z    +0.000, E1  +303.950, E3 -233801.008}
SPL {X  -121.335, Y  +278.219, Z    +0.000, E1  +311.699, E3 -233899.355}
ENDSPLINE

SPLINE
SPL {X  -146.770, Y  +318.818, Z    +0.000, E1  +325.496, E3 -233999.188}
SPL {X  -156.430, Y  +348.936, Z    +0.000, E1  +338.153, E3 -234015.920}
SPL {X  -159.088, Y  +365.539, Z    +0.000, E1  +347.196, E3 -234020.330}
SPL {X  -159.921, Y  +377.798, Z    +0.000, E1  +354.872, E3 -234021.991}
SPL {X  -159.990, Y  +384.169, Z    +0.000, E1  +359.534, E3 -234022.346}
SPL {X  -159.990, Y  +387.385, Z    +0.000, E1  +362.811, E3 -234022.465}
SPL {X  -159.990, Y  +391.439, Z    +0.000, E1  +368.259, E3 -234022.761}
SPL {X  -159.990, Y  +395.747, Z    +0.000, E1  +374.484, E3 -234023.282}
SPL {X  -159.990, Y  +402.387, Z    +0.000, E1  +384.140, E3 -234024.514}
SPL {X  -159.990, Y  +414.244, Z    +0.000, E1  +397.704, E3 -234028.147}
SPL {X  -159.990, Y  +460.468, Z    +0.000, E1  +416.751, E3 -234052.239}
SPL {X  -159.990, Y  +537.348, Z    +0.000, E1  +420.157, E3 -234122.251}
SPL {X  -159.990, Y  +549.907, Z    +0.000, E1  +420.183, E3 -234137.508}
SPL {X  -159.990, Y  +560.677, Z    +0.000, E1  +420.145, E3 -234150.679}
SPL {X  -159.990, Y  +569.073, Z    +0.000, E1  +420.153, E3 -234160.894}
SPL {X  -159.990, Y  +581.828, Z    +0.000, E1  +420.191, E3 -234176.353}
SPL {X  -159.990, Y  +594.125, Z    +0.000, E1  +420.153, E3 -234191.385}
SPL {X  -159.990, Y  +602.716, Z    +0.000, E1  +420.150, E3 -234201.848}
SPL {X  -159.990, Y  +612.205, Z    +0.000, E1  +420.159, E3 -234213.385}
SPL {X  -159.990, Y  +620.604, Z    +0.000, E1  +420.153, E3 -234223.600}
SPL {X  -159.990, Y  +632.106, Z    +0.000, E1  +420.183, E3 -234237.577}
SPL {X  -159.990, Y  +643.341, Z    +0.000, E1  +420.148, E3 -234251.320}
SPL {X  -159.990, Y  +652.098, Z    +0.000, E1  +420.153, E3 -234261.966}
SPL {X  -159.990, Y  +661.466, Z    +0.000, E1  +420.154, E3 -234273.377}
SPL {X  -159.990, Y  +670.781, Z    +0.000, E1  +420.150, E3 -234284.725}
SPL {X  -159.839, Y  +678.445, Z    +0.000, E1  +420.123, E3 -234294.204}
SPL {X  -159.339, Y  +685.922, Z    +0.000, E1  +420.057, E3 -234303.806}
SPL {X  -158.381, Y  +694.132, Z    +0.000, E1  +419.909, E3 -234314.804}
SPL {X  -157.192, Y  +701.291, Z    +0.000, E1  +419.715, E3 -234324.774}
SPL {X  -155.426, Y  +709.440, Z    +0.000, E1  +419.459, E3 -234336.472}
SPL {X  -153.239, Y  +717.485, Z    +0.000, E1  +419.087, E3 -234348.517}
SPL {X  -150.608, Y  +725.483, Z    +0.000, E1  +418.677, E3 -234360.862}
SPL {X  -148.008, Y  +732.249, Z    +0.000, E1  +418.192, E3 -234371.729}
SPL {X  -145.943, Y  +737.055, Z    +0.000, E1  +417.829, E3 -234379.587}
SPL {X  -143.898, Y  +741.430, Z    +0.000, E1  +417.467, E3 -234386.857}
SPL {X  -140.579, Y  +747.882, Z    +0.000, E1  +416.895, E3 -234397.736}
SPL {X  -137.120, Y  +753.931, Z    +0.000, E1  +416.213, E3 -234408.196}
SPL {X  -120.054, Y  +777.254, Z    +0.000, E1  +409.463, E3 -234494.942}
ENDSPLINE

SPLINE
SPL {X  -141.034, Y  +747.040, Z    +0.000, E1  +398.619, E3 -234603.104}
SPL {X  -152.334, Y  +720.400, Z    +0.000, E1  +389.143, E3 -234622.558}
SPL {X  -157.190, Y  +701.303, Z    +0.000, E1  +380.164, E3 -234629.719}
SPL {X  -159.460, Y  +684.516, Z    +0.000, E1  +370.556, E3 -234633.314}
SPL {X  -159.938, Y  +675.597, Z    +0.000, E1  +364.669, E3 -234634.321}
SPL {X  -159.990, Y  +669.975, Z    +0.000, E1  +360.595, E3 -234634.571}
SPL {X  -159.990, Y  +666.850, Z    +0.000, E1  +357.321, E3 -234634.672}
SPL {X  -159.990, Y  +662.495, Z    +0.000, E1  +351.318, E3 -234634.966}
SPL {X  -159.990, Y  +657.714, Z    +0.000, E1  +344.114, E3 -234635.527}
SPL {X  -159.990, Y  +651.822, Z    +0.000, E1  +335.261, E3 -234636.496}
SPL {X  -159.990, Y  +641.369, Z    +0.000, E1  +322.665, E3 -234639.334}
SPL {X  -159.990, Y  +598.251, Z    +0.000, E1  +304.104, E3 -234663.105}
SPL {X  -159.990, Y  +514.954, Z    +0.000, E1  +299.688, E3 -234736.901}
SPL {X  -159.990, Y  +501.679, Z    +0.000, E1  +299.667, E3 -234752.937}
SPL {X  -159.990, Y  +488.988, Z    +0.000, E1  +299.693, E3 -234768.340}
SPL {X  -159.990, Y  +478.987, Z    +0.000, E1  +299.694, E3 -234780.443}
SPL {X  -159.990, Y  +468.796, Z    +0.000, E1  +299.698, E3 -234792.786}
SPL {X  -159.990, Y  +460.399, Z    +0.000, E1  +299.707, E3 -234802.963}
SPL {X  -159.990, Y  +453.289, Z    +0.000, E1  +299.707, E3 -234811.569}
SPL {X  -159.990, Y  +443.890, Z    +0.000, E1  +299.691, E3 -234822.922}
SPL {X  -159.990, Y  +437.910, Z    +0.000, E1  +300.175, E3 -234833.393}
ENDSPLINE

SPLINE
SPL {X  -159.990, Y  +447.165, Z    +0.000, E1  +303.287, E3 -234841.948}
ENDSPLINE

SPLINE
SPL {X  -159.990, Y  +436.354, Z    +0.000, E1  +302.683, E3 -234852.960}
SPL {X  -159.990, Y  +425.140, Z    +0.000, E1  +301.982, E3 -234863.395}
SPL {X  -159.990, Y  +412.625, Z    +0.000, E1  +301.150, E3 -234874.231}
SPL {X  -159.990, Y  +398.951, Z    +0.000, E1  +300.353, E3 -234886.102}
SPL {X  -159.990, Y  +389.564, Z    +0.000, E1  +300.093, E3 -234895.916}
SPL {X  -159.985, Y  +381.230, Z    +0.000, E1  +300.090, E3 -234906.183}
SPL {X  -159.702, Y  +372.900, Z    +0.000, E1  +300.135, E3 -234916.720}
SPL {X  -159.030, Y  +365.001, Z    +0.000, E1  +300.230, E3 -234927.123}
SPL {X  -157.449, Y  +354.098, Z    +0.000, E1  +300.447, E3 -234942.123}
SPL {X  -155.503, Y  +344.875, Z    +0.000, E1  +300.798, E3 -234955.541}
SPL {X  -153.622, Y  +337.813, Z    +0.000, E1  +301.097, E3 -234966.135}
SPL {X  -150.877, Y  +329.275, Z    +0.000, E1  +301.527, E3 -234979.359}
SPL {X  -148.134, Y  +322.059, Z    +0.000, E1  +302.038, E3 -234990.998}
SPL {X  -145.832, Y  +316.699, Z    +0.000, E1  +302.442, E3 -234999.832}
SPL {X  -143.160, Y  +311.071, Z    +0.000, E1  +302.918, E3 -235009.278}
SPL {X  -140.427, Y  +305.839, Z    +0.000, E1  +303.430, E3 -235018.239}
SPL {X  -137.611, Y  +300.891, Z    +0.000, E1  +303.950, E3 -235026.815}
SPL {X  -121.335, Y  +278.219, Z    +0.000, E1  +311.699, E3 -235125.161}
ENDSPLINE

SPLINE
SPL {X  -146.770, Y  +318.818, Z    +0.000, E1  +325.496, E3 -235224.995}
SPL {X  -156.430, Y  +348.936, Z    +0.000, E1  +338.153, E3 -235241.726}
SPL {X  -159.088, Y  +365.539, Z    +0.000, E1  +347.196, E3 -235246.137}
SPL {X  -159.921, Y  +377.798, Z    +0.000, E1  +354.872, E3 -235247.797}
SPL {X  -159.990, Y  +383.148, Z    +0.000, E1  +358.786, E3 -235248.125}
SPL {X  -159.990, Y  +385.595, Z    +0.000, E1  +360.838, E3 -235248.194}
SPL {X  -159.990, Y  +390.176, Z    +0.000, E1  +366.367, E3 -235248.463}
SPL {X  -159.990, Y  +395.747, Z    +0.000, E1  +374.484, E3 -235249.088}
SPL {X  -159.990, Y  +402.387, Z    +0.000, E1  +384.140, E3 -235250.321}
SPL {X  -159.990, Y  +413.408, Z    +0.000, E1  +396.965, E3 -235253.622}
SPL {X  -159.990, Y  +455.723, Z    +0.000, E1  +415.803, E3 -235275.464}
SPL {X  -159.990, Y  +537.348, Z    +0.000, E1  +420.157, E3 -235348.057}
SPL {X  -159.990, Y  +549.907, Z    +0.000, E1  +420.183, E3 -235363.315}
SPL {X  -159.990, Y  +560.677, Z    +0.000, E1  +420.145, E3 -235376.486}
SPL {X  -159.990, Y  +569.073, Z    +0.000, E1  +420.153, E3 -235386.700}
SPL {X  -159.990, Y  +581.828, Z    +0.000, E1  +420.191, E3 -235402.159}
SPL {X  -159.990, Y  +594.125, Z    +0.000, E1  +420.153, E3 -235417.192}
SPL {X  -159.990, Y  +602.716, Z    +0.000, E1  +420.150, E3 -235427.654}
SPL {X  -159.990, Y  +612.205, Z    +0.000, E1  +420.159, E3 -235439.191}
SPL {X  -159.990, Y  +620.604, Z    +0.000, E1  +420.153, E3 -235449.407}
SPL {X  -159.990, Y  +632.106, Z    +0.000, E1  +420.183, E3 -235463.383}
SPL {X  -159.990, Y  +643.341, Z    +0.000, E1  +420.148, E3 -235477.127}
SPL {X  -159.990, Y  +652.098, Z    +0.000, E1  +420.153, E3 -235487.772}
SPL {X  -159.990, Y  +661.466, Z    +0.000, E1  +420.154, E3 -235499.183}
SPL {X  -159.963, Y  +674.441, Z    +0.000, E1  +420.189, E3 -235514.934}
SPL {X  -159.339, Y  +685.922, Z    +0.000, E1  +420.057, E3 -235529.613}
SPL {X  -158.381, Y  +694.132, Z    +0.000, E1  +419.909, E3 -235540.610}
SPL {X  -156.712, Y  +703.719, Z    +0.000, E1  +419.674, E3 -235553.975}
SPL {X  -154.922, Y  +711.450, Z    +0.000, E1  +419.348, E3 -235565.291}
SPL {X  -153.239, Y  +717.485, Z    +0.000, E1  +419.087, E3 -235574.323}
SPL {X  -150.608, Y  +725.483, Z    +0.000, E1  +418.677, E3 -235586.669}
SPL {X  -148.008, Y  +732.249, Z    +0.000, E1  +418.192, E3 -235597.535}
SPL {X  -145.943, Y  +737.055, Z    +0.000, E1  +417.829, E3 -235605.394}
SPL {X  -143.898, Y  +741.430, Z    +0.000, E1  +417.467, E3 -235612.663}
SPL {X  -141.624, Y  +745.927, Z    +0.000, E1  +417.045, E3 -235620.259}
SPL {X  -139.581, Y  +749.692, Z    +0.000, E1  +416.662, E3 -235626.705}
SPL {X  -137.120, Y  +753.931, Z    +0.000, E1  +416.213, E3 -235634.002}
SPL {X  -120.054, Y  +777.254, Z    +0.000, E1  +409.463, E3 -235720.748}
ENDSPLINE

SPLINE
SPL {X  -141.034, Y  +747.040, Z    +0.000, E1  +398.619, E3 -235828.910}
SPL {X  -152.334, Y  +720.400, Z    +0.000, E1  +389.143, E3 -235848.365}
SPL {X  -157.190, Y  +701.303, Z    +0.000, E1  +380.164, E3 -235855.525}
SPL {X  -159.460, Y  +684.516, Z    +0.000, E1  +370.556, E3 -235859.121}
SPL {X  -159.938, Y  +675.597, Z    +0.000, E1  +364.669, E3 -235860.127}
SPL {X  -159.990, Y  +669.975, Z    +0.000, E1  +360.595, E3 -235860.378}
SPL {X  -159.990, Y  +666.850, Z    +0.000, E1  +357.321, E3 -235860.478}
SPL {X  -159.990, Y  +662.495, Z    +0.000, E1  +351.318, E3 -235860.773}
SPL {X  -159.990, Y  +657.714, Z    +0.000, E1  +344.114, E3 -235861.334}
SPL {X  -159.990, Y  +651.822, Z    +0.000, E1  +335.261, E3 -235862.302}
SPL {X  -159.990, Y  +641.369, Z    +0.000, E1  +322.665, E3 -235865.140}
SPL {X  -159.990, Y  +598.251, Z    +0.000, E1  +304.104, E3 -235888.912}
SPL {X  -159.990, Y  +514.954, Z    +0.000, E1  +299.688, E3 -235962.707}
SPL {X  -159.990, Y  +505.641, Z    +0.000, E1  +299.707, E3 -235974.016}
SPL {X  -159.990, Y  +498.210, Z    +0.000, E1  +299.707, E3 -235983.010}
SPL {X  -159.990, Y  +488.988, Z    +0.000, E1  +299.693, E3 -235994.146}
SPL {X  -159.990, Y  +478.987, Z    +0.000, E1  +299.694, E3 -236006.249}
SPL {X  -159.990, Y  +468.796, Z    +0.000, E1  +299.698, E3 -236018.593}
SPL {X  -159.990, Y  +460.399, Z    +0.000, E1  +299.707, E3 -236028.770}
SPL {X  -159.990, Y  +453.289, Z    +0.000, E1  +299.707, E3 -236037.375}
SPL {X  -159.990, Y  +443.890, Z    +0.000, E1  +299.691, E3 -236048.729}
SPL {X  -159.990, Y  +437.910, Z    +0.000, E1  +300.175, E3 -236059.199}
ENDSPLINE

SPLINE
SPL {X  -159.990, Y  +447.165, Z    +0.000, E1  +303.287, E3 -236067.755}
ENDSPLINE

SPLINE
SPL {X  -159.990, Y  +436.354, Z    +0.000, E1  +302.683, E3 -236078.766}
SPL {X  -159.990, Y  +425.140, Z    +0.000, E1  +301.982, E3 -236089.201}
SPL {X  -159.990, Y  +412.625, Z    +0.000, E1  +301.150, E3 -236100.038}
SPL {X  -159.990, Y  +398.951, Z    +0.000, E1  +300.353, E3 -236111.909}
SPL {X  -159.990, Y  +389.564, Z    +0.000, E1  +300.093, E3 -236121.723}
SPL {X  -159.985, Y  +381.230, Z    +0.000, E1  +300.090, E3 -236131.990}
SPL {X  -159.702, Y  +372.900, Z    +0.000, E1  +300.135, E3 -236142.527}
SPL {X  -159.030, Y  +365.001, Z    +0.000, E1  +300.230, E3 -236152.930}
SPL {X  -157.449, Y  +354.098, Z    +0.000, E1  +300.447, E3 -236167.929}
SPL {X  -155.503, Y  +344.875, Z    +0.000, E1  +300.798, E3 -236181.348}
SPL {X  -153.622, Y  +337.813, Z    +0.000, E1  +301.097, E3 -236191.941}
SPL {X  -150.877, Y  +329.275, Z    +0.000, E1  +301.527, E3 -236205.166}
SPL {X  -148.134, Y  +322.059, Z    +0.000, E1  +302.038, E3 -236216.804}
SPL {X  -145.832, Y  +316.699, Z    +0.000, E1  +302.442, E3 -236225.639}
SPL {X  -143.160, Y  +311.071, Z    +0.000, E1  +302.918, E3 -236235.084}
SPL {X  -140.427, Y  +305.839, Z    +0.000, E1  +303.430, E3 -236244.045}
SPL {X  -137.611, Y  +300.891, Z    +0.000, E1  +303.950, E3 -236252.621}
SPL {X  -121.335, Y  +278.219, Z    +0.000, E1  +311.699, E3 -236350.967}
ENDSPLINE

SPLINE
SPL {X  -146.770, Y  +318.818, Z    +0.000, E1  +325.496, E3 -236450.801}
SPL {X  -156.430, Y  +348.936, Z    +0.000, E1  +338.153, E3 -236467.533}
SPL {X  -159.088, Y  +365.539, Z    +0.000, E1  +347.196, E3 -236471.943}
SPL {X  -159.820, Y  +375.127, Z    +0.000, E1  +353.170, E3 -236473.367}
SPL {X  -159.990, Y  +382.134, Z    +0.000, E1  +357.935, E3 -236473.886}
SPL {X  -159.990, Y  +385.595, Z    +0.000, E1  +360.838, E3 -236474.000}
SPL {X  -159.990, Y  +390.176, Z    +0.000, E1  +366.367, E3 -236474.269}
SPL {X  -159.990, Y  +395.747, Z    +0.000, E1  +374.484, E3 -236474.895}
SPL {X  -159.990, Y  +404.190, Z    +0.000, E1  +386.444, E3 -236476.577}
SPL {X  -159.990, Y  +418.143, Z    +0.000, E1  +401.167, E3 -236481.170}
SPL {X  -159.990, Y  +460.468, Z    +0.000, E1  +416.751, E3 -236503.852}
SPL {X  -159.990, Y  +537.348, Z    +0.000, E1  +420.157, E3 -236573.863}
SPL {X  -159.990, Y  +549.907, Z    +0.000, E1  +420.183, E3 -236589.121}
SPL {X  -159.990, Y  +560.677, Z    +0.000, E1  +420.145, E3 -236602.292}
SPL {X  -159.990, Y  +569.073, Z    +0.000, E1  +420.153, E3 -236612.506}
SPL {X  -159.990, Y  +581.828, Z    +0.000, E1  +420.191, E3 -236627.966}
SPL {X  -159.990, Y  +594.125, Z    +0.000, E1  +420.153, E3 -236642.998}
SPL {X  -159.990, Y  +602.716, Z    +0.000, E1  +420.150, E3 -236653.461}
SPL {X  -159.990, Y  +612.205, Z    +0.000, E1  +420.159, E3 -236664.997}
SPL {X  -159.990, Y  +620.604, Z    +0.000, E1  +420.153, E3 -236675.213}
SPL {X  -159.990, Y  +632.106, Z    +0.000, E1  +420.183, E3 -236689.190}
SPL {X  -159.990, Y  +643.341, Z    +0.000, E1  +420.148, E3 -236702.933}
SPL {X  -159.990, Y  +652.098, Z    +0.000, E1  +420.153, E3 -236713.579}
SPL {X  -159.990, Y  +661.466, Z    +0.000, E1  +420.154, E3 -236724.990}
SPL {X  -159.990, Y  +670.781, Z    +0.000, E1  +420.150, E3 -236736.338}
SPL {X  -159.839, Y  +678.445, Z    +0.000, E1  +420.123, E3 -236745.817}
SPL {X  -159.339, Y  +685.922, Z    +0.000, E1  +420.057, E3 -236755.419}
SPL {X  -158.381, Y  +694.132, Z    +0.000, E1  +419.909, E3 -236766.416}
SPL {X  -157.192, Y  +701.291, Z    +0.000, E1  +419.715, E3 -236776.387}
SPL {X  -155.426, Y  +709.440, Z    +0.000, E1  +419.459, E3 -236788.085}
SPL {X  -153.239, Y  +717.485, Z    +0.000, E1  +419.087, E3 -236800.130}
SPL {X  -150.608, Y  +725.483, Z    +0.000, E1  +418.677, E3 -236812.475}
SPL {X  -148.008, Y  +732.249, Z    +0.000, E1  +418.192, E3 -236823.342}
SPL {X  -145.943, Y  +737.055, Z    +0.000, E1  +417.829, E3 -236831.200}
SPL {X  -143.898, Y  +741.430, Z    +0.000, E1  +417.467, E3 -236838.470}
SPL {X  -141.624, Y  +745.927, Z    +0.000, E1  +417.045, E3 -236846.065}
SPL {X  -139.581, Y  +749.692, Z    +0.000, E1  +416.662, E3 -236852.512}
SPL {X  -137.120, Y  +753.931, Z    +0.000, E1  +416.213, E3 -236859.809}
SPL {X  -120.054, Y  +777.254, Z    +0.000, E1  +409.463, E3 -236946.555}
ENDSPLINE

SPLINE
SPL {X  -141.034, Y  +747.040, Z    +0.000, E1  +398.619, E3 -237054.717}
SPL {X  -152.334, Y  +720.400, Z    +0.000, E1  +389.143, E3 -237074.171}
SPL {X  -157.190, Y  +701.303, Z    +0.000, E1  +380.164, E3 -237081.332}
SPL {X  -159.460, Y  +684.516, Z    +0.000, E1  +370.556, E3 -237084.927}
SPL {X  -159.938, Y  +675.597, Z    +0.000, E1  +364.669, E3 -237085.934}
SPL {X  -159.990, Y  +671.043, Z    +0.000, E1  +361.371, E3 -237086.157}
SPL {X  -159.990, Y  +669.269, Z    +0.000, E1  +359.855, E3 -237086.202}
SPL {X  -159.990, Y  +666.850, Z    +0.000, E1  +357.321, E3 -237086.285}
SPL {X  -159.990, Y  +662.495, Z    +0.000, E1  +351.318, E3 -237086.579}
SPL {X  -159.990, Y  +657.714, Z    +0.000, E1  +344.114, E3 -237087.140}
SPL {X  -159.990, Y  +651.822, Z    +0.000, E1  +335.261, E3 -237088.108}
SPL {X  -159.990, Y  +641.369, Z    +0.000, E1  +322.665, E3 -237090.947}
SPL {X  -159.990, Y  +598.251, Z    +0.000, E1  +304.104, E3 -237114.718}
SPL {X  -159.990, Y  +514.954, Z    +0.000, E1  +299.688, E3 -237188.513}
SPL {X  -159.990, Y  +505.641, Z    +0.000, E1  +299.707, E3 -237199.823}
SPL {X  -159.990, Y  +498.210, Z    +0.000, E1  +299.707, E3 -237208.816}
SPL {X  -159.990, Y  +488.988, Z    +0.000, E1  +299.693, E3 -237219.953}
SPL {X  -159.990, Y  +478.987, Z    +0.000, E1  +299.694, E3 -237232.055}
SPL {X  -159.990, Y  +468.796, Z    +0.000, E1  +299.698, E3 -237244.399}
SPL {X  -159.990, Y  +456.606, Z    +0.000, E1  +299.670, E3 -237259.105}
SPL {X  -159.990, Y  +443.890, Z    +0.000, E1  +299.691, E3 -237274.535}
SPL {X  -159.990, Y  +437.910, Z    +0.000, E1  +300.175, E3 -237285.006}
ENDSPLINE

SPLINE
SPL {X  -159.990, Y  +447.165, Z    +0.000, E1  +303.287, E3 -237293.561}
ENDSPLINE

SPLINE
SPL {X  -159.990, Y  +436.354, Z    +0.000, E1  +302.683, E3 -237304.572}
SPL {X  -159.990, Y  +425.140, Z    +0.000, E1  +301.982, E3 -237315.008}
SPL {X  -159.990, Y  +412.625, Z    +0.000, E1  +301.150, E3 -237325.844}
SPL {X  -159.990, Y  +398.951, Z    +0.000, E1  +300.353, E3 -237337.715}
SPL {X  -159.990, Y  +389.564, Z    +0.000, E1  +300.093, E3 -237347.529}
SPL {X  -159.985, Y  +381.230, Z    +0.000, E1  +300.090, E3 -237357.796}
SPL {X  -159.702, Y  +372.900, Z    +0.000, E1  +300.135, E3 -237368.333}
SPL {X  -159.030, Y  +365.001, Z    +0.000, E1  +300.230, E3 -237378.736}
SPL {X  -158.029, Y  +357.528, Z    +0.000, E1  +300.403, E3 -237388.991}
SPL {X  -156.953, Y  +351.476, Z    +0.000, E1  +300.570, E3 -237397.545}
SPL {X  -155.503, Y  +344.875, Z    +0.000, E1  +300.798, E3 -237407.154}
SPL {X  -153.622, Y  +337.813, Z    +0.000, E1  +301.097, E3 -237417.748}
SPL {X  -150.877, Y  +329.275, Z    +0.000, E1  +301.527, E3 -237430.972}
SPL {X  -148.134, Y  +322.059, Z    +0.000, E1  +302.038, E3 -237442.611}
SPL {X  -145.832, Y  +316.699, Z    +0.000, E1  +302.442, E3 -237451.445}
SPL {X  -143.160, Y  +311.071, Z    +0.000, E1  +302.918, E3 -237460.891}
SPL {X  -140.427, Y  +305.839, Z    +0.000, E1  +303.430, E3 -237469.852}
SPL {X  -137.611, Y  +300.891, Z    +0.000, E1  +303.950, E3 -237478.428}
SPL {X  -121.335, Y  +278.219, Z    +0.000, E1  +311.699, E3 -237576.774}
ENDSPLINE

SPLINE
SPL {X  -146.770, Y  +318.818, Z    +0.000, E1  +325.496, E3 -237676.608}
SPL {X  -156.430, Y  +348.936, Z    +0.000, E1  +338.153, E3 -237693.339}
SPL {X  -159.088, Y  +365.539, Z    +0.000, E1  +347.196, E3 -237697.750}
SPL {X  -159.921, Y  +377.798, Z    +0.000, E1  +354.872, E3 -237699.410}
SPL {X  -159.990, Y  +384.169, Z    +0.000, E1  +359.534, E3 -237699.766}
SPL {X  -159.990, Y  +386.366, Z    +0.000, E1  +361.774, E3 -237699.830}
SPL {X  -159.990, Y  +390.176, Z    +0.000, E1  +366.367, E3 -237700.076}
SPL {X  -159.990, Y  +395.747, Z    +0.000, E1  +374.484, E3 -237700.701}
SPL {X  -159.990, Y  +402.387, Z    +0.000, E1  +384.140, E3 -237701.934}
SPL {X  -159.990, Y  +414.244, Z    +0.000, E1  +397.704, E3 -237705.567}
SPL {X  -159.990, Y  +460.468, Z    +0.000, E1  +416.751, E3 -237729.658}
SPL {X  -159.990, Y  +537.348, Z    +0.000, E1  +420.157, E3 -237799.670}
SPL {X  -159.990, Y  +545.972, Z    +0.000, E1  +420.143, E3 -237810.204}
SPL {X  -159.990, Y  +557.131, Z    +0.000, E1  +420.184, E3 -237823.718}
SPL {X  -159.990, Y  +569.073, Z    +0.000, E1  +420.153, E3 -237838.313}
SPL {X  -159.990, Y  +581.828, Z    +0.000, E1  +420.191, E3 -237853.772}
SPL {X  -159.990, Y  +594.125, Z    +0.000, E1  +420.153, E3 -237868.805}
SPL {X  -159.990, Y  +602.716, Z    +0.000, E1  +420.150, E3 -237879.267}
SPL {X  -159.990, Y  +612.205, Z    +0.000, E1  +420.159, E3 -237890.804}
SPL {X  -159.990, Y  +624.752, Z    +0.000, E1  +420.194, E3 -237906.012}
SPL {X  -159.990, Y  +640.062, Z    +0.000, E1  +420.188, E3 -237924.675}
SPL {X  -159.990, Y  +652.098, Z    +0.000, E1  +420.153, E3 -237939.385}
SPL {X  -159.990, Y  +661.466, Z    +0.000, E1  +420.154, E3 -237950.796}
SPL {X  -159.963, Y  +674.441, Z    +0.000, E1  +420.189, E3 -237966.547}
SPL {X  -159.339, Y  +685.922, Z    +0.000, E1  +420.057, E3 -237981.226}
SPL {X  -158.381, Y  +694.132, Z    +0.000, E1  +419.909, E3 -237992.223}
SPL {X  -156.712, Y  +703.719, Z    +0.000, E1  +419.674, E3 -238005.588}
SPL {X  -154.922, Y  +711.450, Z    +0.000, E1  +419.348, E3 -238016.904}
SPL {X  -153.239, Y  +717.485, Z    +0.000, E1  +419.087, E3 -238025.936}
SPL {X  -150.608, Y  +725.483, Z    +0.000, E1  +418.677, E3 -238038.282}
SPL {X  -148.008, Y  +732.249, Z    +0.000, E1  +418.192, E3 -238049.148}
SPL {X  -145.943, Y  +737.055, Z    +0.000, E1  +417.829, E3 -238057.007}
SPL {X  -143.898, Y  +741.430, Z    +0.000, E1  +417.467, E3 -238064.276}
SPL {X  -141.624, Y  +745.927, Z    +0.000, E1  +417.045, E3 -238071.871}
SPL {X  -139.581, Y  +749.692, Z    +0.000, E1  +416.662, E3 -238078.318}
SPL {X  -137.120, Y  +753.931, Z    +0.000, E1  +416.213, E3 -238085.615}
SPL {X  -120.054, Y  +777.254, Z    +0.000, E1  +409.463, E3 -238172.361}
ENDSPLINE

SPLINE
SPL {X  -141.034, Y  +747.040, Z    +0.000, E1  +398.619, E3 -238280.523}
SPL {X  -152.334, Y  +720.400, Z    +0.000, E1  +389.143, E3 -238299.977}
SPL {X  -157.190, Y  +701.303, Z    +0.000, E1  +380.164, E3 -238307.138}
SPL {X  -159.117, Y  +688.191, Z    +0.000, E1  +372.748, E3 -238310.170}
SPL {X  -159.875, Y  +677.561, Z    +0.000, E1  +366.083, E3 -238311.560}
SPL {X  -159.990, Y  +669.975, Z    +0.000, E1  +360.595, E3 -238311.991}
SPL {X  -159.990, Y  +666.850, Z    +0.000, E1  +357.321, E3 -238312.091}
SPL {X  -159.990, Y  +662.495, Z    +0.000, E1  +351.318, E3 -238312.386}
SPL {X  -159.990, Y  +657.714, Z    +0.000, E1  +344.114, E3 -238312.947}
SPL {X  -159.990, Y  +651.822, Z    +0.000, E1  +335.261, E3 -238313.915}
SPL {X  -159.990, Y  +641.369, Z    +0.000, E1  +322.665, E3 -238316.753}
SPL {X  -159.990, Y  +598.251, Z    +0.000, E1  +304.104, E3 -238340.524}
SPL {X  -159.990, Y  +514.954, Z    +0.000, E1  +299.688, E3 -238414.320}
SPL {X  -159.990, Y  +505.641, Z    +0.000, E1  +299.707, E3 -238425.629}
SPL {X  -159.990, Y  +498.210, Z    +0.000, E1  +299.707, E3 -238434.623}
SPL {X  -159.990, Y  +488.988, Z    +0.000, E1  +299.693, E3 -238445.759}
SPL {X  -159.990, Y  +478.987, Z    +0.000, E1  +299.694, E3 -238457.862}
SPL {X  -159.990, Y  +468.796, Z    +0.000, E1  +299.698, E3 -238470.206}
SPL {X  -159.990, Y  +460.399, Z    +0.000, E1  +299.707, E3 -238480.382}
SPL {X  -159.990, Y  +453.289, Z    +0.000, E1  +299.707, E3 -238488.988}
SPL {X  -159.990, Y  +443.890, Z    +0.000, E1  +299.691, E3 -238500.341}
SPL {X  -159.990, Y  +437.910, Z    +0.000, E1  +300.175, E3 -238510.812}
ENDSPLINE

SPLINE
SPL {X  -159.990, Y  +447.165, Z    +0.000, E1  +303.287, E3 -238519.367}
ENDSPLINE

SPLINE
SPL {X  -159.990, Y  +436.354, Z    +0.000, E1  +302.683, E3 -238530.379}
SPL {X  -159.990, Y  +425.140, Z    +0.000, E1  +301.982, E3 -238540.814}
SPL {X  -159.990, Y  +412.625, Z    +0.000, E1  +301.150, E3 -238551.650}
SPL {X  -159.990, Y  +398.951, Z    +0.000, E1  +300.353, E3 -238563.522}
SPL {X  -159.990, Y  +389.564, Z    +0.000, E1  +300.093, E3 -238573.336}
SPL {X  -159.985, Y  +381.230, Z    +0.000, E1  +300.090, E3 -238583.603}
SPL {X  -159.702, Y  +372.900, Z    +0.000, E1  +300.135, E3 -238594.140}
SPL {X  -159.030, Y  +365.001, Z    +0.000, E1  +300.230, E3 -238604.542}
SPL {X  -157.449, Y  +354.098, Z    +0.000, E1  +300.447, E3 -238619.542}
SPL {X  -155.503, Y  +344.875, Z    +0.000, E1  +300.798, E3 -238632.961}
SPL {X  -153.622, Y  +337.813, Z    +0.000, E1  +301.097, E3 -238643.554}
SPL {X  -150.877, Y  +329.275, Z    +0.000, E1  +301.527, E3 -238656.779}
SPL {X  -148.134, Y  +322.059, Z    +0.000, E1  +302.038, E3 -238668.417}
SPL {X  -145.832, Y  +316.699, Z    +0.000, E1  +302.442, E3 -238677.252}
SPL {X  -143.160, Y  +311.071, Z    +0.000, E1  +302.918, E3 -238686.697}
SPL {X  -139.570, Y  +304.288, Z    +0.000, E1  +303.552, E3 -238698.293}
SPL {X  -136.734, Y  +299.430, Z    +0.000, E1  +304.147, E3 -238706.832}
SPL {X  -121.335, Y  +278.219, Z    +0.000, E1  +311.699, E3 -238802.580}
ENDSPLINE

SPLINE
SPL {X  -146.770, Y  +318.818, Z    +0.000, E1  +325.496, E3 -238902.414}
SPL {X  -156.430, Y  +348.936, Z    +0.000, E1  +338.153, E3 -238919.145}
SPL {X  -159.088, Y  +365.539, Z    +0.000, E1  +347.196, E3 -238923.556}
SPL {X  -159.921, Y  +377.798, Z    +0.000, E1  +354.872, E3 -238925.216}
SPL {X  -159.990, Y  +384.169, Z    +0.000, E1  +359.534, E3 -238925.572}
SPL {X  -159.990, Y  +387.385, Z    +0.000, E1  +362.811, E3 -238925.691}
SPL {X  -159.990, Y  +391.439, Z    +0.000, E1  +368.259, E3 -238925.987}
SPL {X  -159.990, Y  +395.747, Z    +0.000, E1  +374.484, E3 -238926.508}
SPL {X  -159.990, Y  +402.387, Z    +0.000, E1  +384.140, E3 -238927.740}
SPL {X  -159.990, Y  +413.408, Z    +0.000, E1  +396.965, E3 -238931.041}
SPL {X  -159.990, Y  +455.723, Z    +0.000, E1  +415.803, E3 -238952.884}
SPL {X  -159.990, Y  +537.348, Z    +0.000, E1  +420.157, E3 -239025.476}
SPL {X  -159.990, Y  +545.972, Z    +0.000, E1  +420.143, E3 -239036.010}
SPL {X  -159.990, Y  +557.131, Z    +0.000, E1  +420.184, E3 -239049.525}
SPL {X  -159.990, Y  +569.073, Z    +0.000, E1  +420.153, E3 -239064.119}
SPL {X  -159.990, Y  +577.562, Z    +0.000, E1  +420.146, E3 -239074.459}
SPL {X  -159.990, Y  +585.415, Z    +0.000, E1  +420.147, E3 -239084.025}
SPL {X  -159.990, Y  +594.125, Z    +0.000, E1  +420.153, E3 -239094.611}
SPL {X  -159.990, Y  +602.716, Z    +0.000, E1  +420.150, E3 -239105.074}
SPL {X  -159.990, Y  +612.205, Z    +0.000, E1  +420.159, E3 -239116.610}
SPL {X  -159.990, Y  +624.752, Z    +0.000, E1  +420.194, E3 -239131.818}
SPL {X  -159.990, Y  +640.062, Z    +0.000, E1  +420.188, E3 -239150.482}
SPL {X  -159.990, Y  +652.098, Z    +0.000, E1  +420.153, E3 -239165.191}
SPL {X  -159.990, Y  +661.466, Z    +0.000, E1  +420.154, E3 -239176.603}
SPL {X  -159.963, Y  +674.441, Z    +0.000, E1  +420.189, E3 -239192.353}
SPL {X  -159.339, Y  +685.922, Z    +0.000, E1  +420.057, E3 -239207.032}
SPL {X  -158.381, Y  +694.132, Z    +0.000, E1  +419.909, E3 -239218.029}
SPL {X  -157.192, Y  +701.291, Z    +0.000, E1  +419.715, E3 -239228.000}
SPL {X  -155.426, Y  +709.440, Z    +0.000, E1  +419.459, E3 -239239.698}
SPL {X  -153.239, Y  +717.485, Z    +0.000, E1  +419.087, E3 -239251.743}
SPL {X  -150.608, Y  +725.483, Z    +0.000, E1  +418.677, E3 -239264.088}
SPL {X  -148.008, Y  +732.249, Z    +0.000, E1  +418.192, E3 -239274.955}
SPL {X  -145.943, Y  +737.055, Z    +0.000, E1  +417.829, E3 -239282.813}
SPL {X  -143.898, Y  +741.430, Z    +0.000, E1  +417.467, E3 -239290.083}
SPL {X  -140.579, Y  +747.882, Z    +0.000, E1  +416.895, E3 -239300.962}
SPL {X  -137.120, Y  +753.931, Z    +0.000, E1  +416.213, E3 -239311.422}
SPL {X  -120.054, Y  +777.254, Z    +0.000, E1  +409.463, E3 -239398.168}
ENDSPLINE

SPLINE
SPL {X  -141.034, Y  +747.040, Z    +0.000, E1  +398.619, E3 -239506.330}
SPL {X  -152.334, Y  +720.400, Z    +0.000, E1  +389.143, E3 -239525.784}
SPL {X  -157.190, Y  +701.303, Z    +0.000, E1  +380.164, E3 -239532.945}
SPL {X  -159.117, Y  +688.191, Z    +0.000, E1  +372.748, E3 -239535.977}
SPL {X  -159.875, Y  +677.561, Z    +0.000, E1  +366.083, E3 -239537.366}
SPL {X  -159.990, Y  +671.043, Z    +0.000, E1  +361.371, E3 -239537.770}
SPL {X  -159.990, Y  +669.269, Z    +0.000, E1  +359.855, E3 -239537.815}
SPL {X  -159.990, Y  +666.850, Z    +0.000, E1  +357.321, E3 -239537.897}
SPL {X  -159.990, Y  +662.495, Z    +0.000, E1  +351.318, E3 -239538.192}
SPL {X  -159.990, Y  +657.714, Z    +0.000, E1  +344.114, E3 -239538.753}
SPL {X  -159.990, Y  +651.822, Z    +0.000, E1  +335.261, E3 -239539.721}
SPL {X  -159.990, Y  +641.369, Z    +0.000, E1  +322.665, E3 -239542.560}
SPL {X  -159.990, Y  +598.251, Z    +0.000, E1  +304.104, E3 -239566.331}
SPL {X  -159.990, Y  +514.954, Z    +0.000, E1  +299.688, E3 -239640.126}
SPL {X  -159.990, Y  +505.641, Z    +0.000, E1  +299.707, E3 -239651.435}
SPL {X  -159.990, Y  +498.210, Z    +0.000, E1  +299.707, E3 -239660.429}
SPL {X  -159.990, Y  +488.988, Z    +0.000, E1  +299.693, E3 -239671.566}
SPL {X  -159.990, Y  +478.987, Z    +0.000, E1  +299.694, E3 -239683.668}
SPL {X  -159.990, Y  +468.796, Z    +0.000, E1  +299.698, E3 -239696.012}
SPL {X  -159.990, Y  +460.399, Z    +0.000, E1  +299.707, E3 -239706.189}
SPL {X  -159.990, Y  +453.289, Z    +0.000, E1  +299.707, E3 -239714.794}
SPL {X  -159.990, Y  +443.890, Z    +0.000, E1  +299.691, E3 -239726.148}
SPL {X  -159.990, Y  +437.910, Z    +0.000, E1  +300.175, E3 -239736.619}
ENDSPLINE

SPLINE
SPL {X  -159.990, Y  +447.165, Z    +0.000, E1  +303.287, E3 -239745.174}
ENDSPLINE

SPLINE
SPL {X  -159.990, Y  +436.354, Z    +0.000, E1  +302.683, E3 -239756.185}
SPL {X  -159.990, Y  +425.140, Z    +0.000, E1  +301.982, E3 -239766.621}
SPL {X  -159.990, Y  +412.625, Z    +0.000, E1  +301.150, E3 -239777.457}
SPL {X  -159.990, Y  +398.951, Z    +0.000, E1  +300.353, E3 -239789.328}
SPL {X  -159.990, Y  +389.564, Z    +0.000, E1  +300.093, E3 -239799.142}
SPL {X  -159.985, Y  +381.230, Z    +0.000, E1  +300.090, E3 -239809.409}
SPL {X  -159.702, Y  +372.900, Z    +0.000, E1  +300.135, E3 -239819.946}
SPL {X  -159.030, Y  +365.001, Z    +0.000, E1  +300.230, E3 -239830.349}
SPL {X  -158.029, Y  +357.528, Z    +0.000, E1  +300.403, E3 -239840.604}
SPL {X  -156.953, Y  +351.476, Z    +0.000, E1  +300.570, E3 -239849.157}
SPL {X  -155.503, Y  +344.875, Z    +0.000, E1  +300.798, E3 -239858.767}
SPL {X  -153.622, Y  +337.813, Z    +0.000, E1  +301.097, E3 -239869.360}
SPL {X  -151.786, Y  +331.925, Z    +0.000, E1  +301.419, E3 -239878.481}
SPL {X  -150.141, Y  +327.233, Z    +0.000, E1  +301.695, E3 -239885.890}
SPL {X  -148.134, Y  +322.059, Z    +0.000, E1  +302.038, E3 -239894.224}
SPL {X  -145.832, Y  +316.699, Z    +0.000, E1  +302.442, E3 -239903.058}
SPL {X  -143.160, Y  +311.071, Z    +0.000, E1  +302.918, E3 -239912.503}
SPL {X  -140.427, Y  +305.839, Z    +0.000, E1  +303.430, E3 -239921.465}
SPL {X  -137.611, Y  +300.891, Z    +0.000, E1  +303.950, E3 -239930.041}
SPL {X  -121.335, Y  +278.219, Z    +0.000, E1  +311.699, E3 -240028.387}
ENDSPLINE

SPLINE
SPL {X  -146.770, Y  +318.818, Z    +0.000, E1  +325.496, E3 -240128.221}
SPL {X  -156.430, Y  +348.936, Z    +0.000, E1  +338.153, E3 -240144.952}
SPL {X  -159.088, Y  +365.539, Z    +0.000, E1  +347.196, E3 -240149.363}
SPL {X  -159.921, Y  +377.798, Z    +0.000, E1  +354.872, E3 -240151.023}
SPL {X  -159.990, Y  +383.148, Z    +0.000, E1  +358.786, E3 -240151.350}
SPL {X  -159.990, Y  +384.761, Z    +0.000, E1  +360.138, E3 -240151.395}
SPL {X  -159.990, Y  +387.385, Z    +0.000, E1  +362.811, E3 -240151.497}
SPL {X  -159.990, Y  +391.439, Z    +0.000, E1  +368.259, E3 -240151.793}
SPL {X  -159.990, Y  +395.747, Z    +0.000, E1  +374.484, E3 -240152.314}
SPL {X  -159.990, Y  +402.387, Z    +0.000, E1  +384.140, E3 -240153.547}
SPL {X  -159.990, Y  +414.244, Z    +0.000, E1  +397.704, E3 -240157.180}
SPL {X  -159.990, Y  +460.468, Z    +0.000, E1  +416.751, E3 -240181.271}
SPL {X  -159.990, Y  +537.348, Z    +0.000, E1  +420.157, E3 -240251.283}
SPL {X  -159.990, Y  +549.907, Z    +0.000, E1  +420.183, E3 -240266.540}
SPL {X  -159.990, Y  +560.677, Z    +0.000, E1  +420.145, E3 -240279.711}
SPL {X  -159.990, Y  +569.073, Z    +0.000, E1  +420.153, E3 -240289.926}
SPL {X  -159.990, Y  +577.562, Z    +0.000, E1  +420.146, E3 -240300.266}
SPL {X  -159.990, Y  +585.415, Z    +0.000, E1  +420.147, E3 -240309.831}
SPL {X  -159.990, Y  +594.125, Z    +0.000, E1  +420.153, E3 -240320.418}
SPL {X  -159.990, Y  +602.716, Z    +0.000, E1  +420.150, E3 -240330.880}
SPL {X  -159.990, Y  +612.205, Z    +0.000, E1  +420.159, E3 -240342.417}
SPL {X  -159.990, Y  +620.604, Z    +0.000, E1  +420.153, E3 -240352.632}
SPL {X  -159.990, Y  +632.106, Z    +0.000, E1  +420.183, E3 -240366.609}
SPL {X  -159.990, Y  +643.341, Z    +0.000, E1  +420.148, E3 -240380.353}
SPL {X  -159.990, Y  +652.098, Z    +0.000, E1  +420.153, E3 -240390.998}
SPL {X  -159.990, Y  +661.466, Z    +0.000, E1  +420.154, E3 -240402.409}
SPL {X  -159.990, Y  +670.781, Z    +0.000, E1  +420.150, E3 -240413.757}
SPL {X  -159.839, Y  +678.445, Z    +0.000, E1  +420.123, E3 -240423.236}
SPL {X  -159.339, Y  +685.922, Z    +0.000, E1  +420.057, E3 -240432.839}
SPL {X  -158.381, Y  +694.132, Z    +0.000, E1  +419.909, E3 -240443.836}
SPL {X  -157.192, Y  +701.291, Z    +0.000, E1  +419.715, E3 -240453.806}
SPL {X  -155.426, Y  +709.440, Z    +0.000, E1  +419.459, E3 -240465.504}
SPL {X  -153.239, Y  +717.485, Z    +0.000, E1  +419.087, E3 -240477.549}
SPL {X  -151.467, Y  +723.022, Z    +0.000, E1  +418.780, E3 -240486.101}
SPL {X  -148.791, Y  +730.306, Z    +0.000, E1  +418.370, E3 -240497.566}
SPL {X  -145.943, Y  +737.055, Z    +0.000, E1  +417.829, E3 -240508.620}
SPL {X  -143.898, Y  +741.430, Z    +0.000, E1  +417.467, E3 -240515.889}
SPL {X  -141.624, Y  +745.927, Z    +0.000, E1  +417.045, E3 -240523.484}
SPL {X  -139.581, Y  +749.692, Z    +0.000, E1  +416.662, E3 -240529.931}
SPL {X  -137.120, Y  +753.931, Z    +0.000, E1  +416.213, E3 -240537.228}
SPL {X  -120.054, Y  +777.254, Z    +0.000, E1  +409.463, E3 -240623.974}
ENDSPLINE

SPLINE
SPL {X  -141.034, Y  +747.040, Z    +0.000, E1  +398.619, E3 -240732.136}
SPL {X  -152.334, Y  +720.400, Z    +0.000, E1  +389.143, E3 -240751.590}
SPL {X  -157.190, Y  +701.303, Z    +0.000, E1  +380.164, E3 -240758.751}
SPL {X  -159.117, Y  +688.191, Z    +0.000, E1  +372.748, E3 -240761.783}
SPL {X  -159.875, Y  +677.561, Z    +0.000, E1  +366.083, E3 -240763.173}
SPL {X  -159.990, Y  +669.975, Z    +0.000, E1  +360.595, E3 -240763.604}
SPL {X  -159.990, Y  +666.850, Z    +0.000, E1  +357.321, E3 -240763.704}
SPL {X  -159.990, Y  +662.495, Z    +0.000, E1  +351.318, E3 -240763.999}
SPL {X  -159.990, Y  +657.714, Z    +0.000, E1  +344.114, E3 -240764.560}
SPL {X  -159.990, Y  +651.822, Z    +0.000, E1  +335.261, E3 -240765.528}
SPL {X  -159.990, Y  +641.369, Z    +0.000, E1  +322.665, E3 -240768.366}
SPL {X  -159.990, Y  +598.251, Z    +0.000, E1  +304.104, E3 -240792.137}
SPL {X  -159.990, Y  +514.954, Z    +0.000, E1  +299.688, E3 -240865.933}
SPL {X  -159.990, Y  +505.641, Z    +0.000, E1  +299.707, E3 -240877.242}
SPL {X  -159.990, Y  +498.210, Z    +0.000, E1  +299.707, E3 -240886.235}
SPL {X  -159.990, Y  +488.988, Z    +0.000, E1  +299.693, E3 -240897.372}
SPL {X  -159.990, Y  +478.987, Z    +0.000, E1  +299.694, E3 -240909.475}
SPL {X  -159.990, Y  +468.796, Z    +0.000, E1  +299.698, E3 -240921.819}
SPL {X  -159.990, Y  +460.399, Z    +0.000, E1  +299.707, E3 -240931.995}
SPL {X  -159.990, Y  +453.289, Z    +0.000, E1  +299.707, E3 -240940.601}
SPL {X  -159.990, Y  +443.890, Z    +0.000, E1  +299.691, E3 -240951.954}
SPL {X  -159.990, Y  +437.910, Z    +0.000, E1  +300.175, E3 -240962.425}
ENDSPLINE

SPLINE
SPL {X  -159.990, Y  +447.165, Z    +0.000, E1  +303.287, E3 -240970.980}
ENDSPLINE

SPLINE
SPL {X  -159.990, Y  +436.354, Z    +0.000, E1  +302.683, E3 -240981.992}
SPL {X  -159.990, Y  +425.140, Z    +0.000, E1  +301.982, E3 -240992.427}
SPL {X  -159.990, Y  +412.625, Z    +0.000, E1  +301.150, E3 -241003.263}
SPL {X  -159.990, Y  +398.951, Z    +0.000, E1  +300.353, E3 -241015.135}
SPL {X  -159.990, Y  +389.564, Z    +0.000, E1  +300.093, E3 -241024.949}
SPL {X  -159.985, Y  +381.230, Z    +0.000, E1  +300.090, E3 -241035.215}
SPL {X  -159.702, Y  +372.900, Z    +0.000, E1  +300.135, E3 -241045.752}
SPL {X  -159.030, Y  +365.001, Z    +0.000, E1  +300.230, E3 -241056.155}
SPL {X  -157.449, Y  +354.098, Z    +0.000, E1  +300.447, E3 -241071.155}
SPL {X  -155.503, Y  +344.875, Z    +0.000, E1  +300.798, E3 -241084.574}
SPL {X  -153.622, Y  +337.813, Z    +0.000, E1  +301.097, E3 -241095.167}
SPL {X  -150.877, Y  +329.275, Z    +0.000, E1  +301.527, E3 -241108.392}
SPL {X  -148.134, Y  +322.059, Z    +0.000, E1  +302.038, E3 -241120.030}
SPL {X  -145.832, Y  +316.699, Z    +0.000, E1  +302.442, E3 -241128.865}
SPL {X  -143.160, Y  +311.071, Z    +0.000, E1  +302.918, E3 -241138.310}
SPL {X  -140.427, Y  +305.839, Z    +0.000, E1  +303.430, E3 -241147.271}
SPL {X  -137.611, Y  +300.891, Z    +0.000, E1  +303.950, E3 -241155.847}
SPL {X  -121.335, Y  +278.219, Z    +0.000, E1  +311.699, E3 -241254.193}
ENDSPLINE

SPLINE
SPL {X  -146.770, Y  +318.818, Z    +0.000, E1  +325.496, E3 -241354.027}
SPL {X  -156.430, Y  +348.936, Z    +0.000, E1  +338.153, E3 -241370.758}
SPL {X  -159.088, Y  +365.539, Z    +0.000, E1  +347.196, E3 -241375.169}
SPL {X  -159.921, Y  +377.798, Z    +0.000, E1  +354.872, E3 -241376.829}
SPL {X  -159.990, Y  +384.169, Z    +0.000, E1  +359.534, E3 -241377.185}
SPL {X  -159.990, Y  +387.385, Z    +0.000, E1  +362.811, E3 -241377.304}
SPL {X  -159.990, Y  +391.439, Z    +0.000, E1  +368.259, E3 -241377.600}
SPL {X  -159.990, Y  +395.747, Z    +0.000, E1  +374.484, E3 -241378.121}
SPL {X  -159.990, Y  +402.387, Z    +0.000, E1  +384.140, E3 -241379.353}
SPL {X  -159.990, Y  +414.244, Z    +0.000, E1  +397.704, E3 -241382.986}
SPL {X  -159.990, Y  +460.468, Z    +0.000, E1  +416.751, E3 -241407.078}
SPL {X  -159.990, Y  +537.348, Z    +0.000, E1  +420.157, E3 -241477.089}
SPL {X  -159.990, Y  +549.907, Z    +0.000, E1  +420.183, E3 -241492.347}
SPL {X  -159.990, Y  +560.677, Z    +0.000, E1  +420.145, E3 -241505.518}
SPL {X  -159.990, Y  +569.073, Z    +0.000, E1  +420.153, E3 -241515.732}
SPL {X  -159.990, Y  +581.828, Z    +0.000, E1  +420.191, E3 -241531.191}
SPL {X  -159.990, Y  +594.125, Z    +0.000, E1  +420.153, E3 -241546.224}
SPL {X  -159.990, Y  +602.716, Z    +0.000, E1  +420.150, E3 -241556.687}
SPL {X  -159.990, Y  +612.205, Z    +0.000, E1  +420.159, E3 -241568.223}
SPL {X  -159.990, Y  +620.604, Z    +0.000, E1  +420.153, E3 -241578.439}
SPL {X  -159.990, Y  +632.106, Z    +0.000, E1  +420.183, E3 -241592.415}
SPL {X  -159.990, Y  +643.341, Z    +0.000, E1  +420.148, E3 -241606.159}
SPL {X  -159.990, Y  +652.098, Z    +0.000, E1  +420.153, E3 -241616.804}
SPL {X  -159.990, Y  +661.466, Z    +0.000, E1  +420.154, E3 -241628.216}
SPL {X  -159.963, Y  +674.441, Z    +0.000, E1  +420.189, E3 -241643.966}
SPL {X  -159.339, Y  +685.922, Z    +0.000, E1  +420.057, E3 -241658.645}
SPL {X  -158.381, Y  +694.132, Z    +0.000, E1  +419.909, E3 -241669.642}
SPL {X  -157.192, Y  +701.291, Z    +0.000, E1  +419.715, E3 -241679.613}
SPL {X  -155.426, Y  +709.440, Z    +0.000, E1  +419.459, E3 -241691.311}
SPL {X  -153.239, Y  +717.485, Z    +0.000, E1  +419.087, E3 -241703.356}
SPL {X  -150.608, Y  +725.483, Z    +0.000, E1  +418.677, E3 -241715.701}
SPL {X  -148.008, Y  +732.249, Z    +0.000, E1  +418.192, E3 -241726.568}
SPL {X  -145.943, Y  +737.055, Z    +0.000, E1  +417.829, E3 -241734.426}
SPL {X  -143.898, Y  +741.430, Z    +0.000, E1  +417.467, E3 -241741.695}
SPL {X  -141.624, Y  +745.927, Z    +0.000, E1  +417.045, E3 -241749.291}
SPL {X  -139.581, Y  +749.692, Z    +0.000, E1  +416.662, E3 -241755.737}
SPL {X  -137.120, Y  +753.931, Z    +0.000, E1  +416.213, E3 -241763.035}
SPL {X  -120.054, Y  +777.254, Z    +0.000, E1  +409.463, E3 -241849.781}
ENDSPLINE

SPLINE
SPL {X  -141.034, Y  +747.040, Z    +0.000, E1  +398.619, E3 -241957.943}
SPL {X  -152.334, Y  +720.400, Z    +0.000, E1  +389.143, E3 -241977.397}
SPL {X  -157.190, Y  +701.303, Z    +0.000, E1  +380.164, E3 -241984.558}
SPL {X  -159.117, Y  +688.191, Z    +0.000, E1  +372.748, E3 -241987.589}
SPL {X  -159.875, Y  +677.561, Z    +0.000, E1  +366.083, E3 -241988.979}
SPL {X  -159.990, Y  +669.975, Z    +0.000, E1  +360.595, E3 -241989.410}
SPL {X  -159.990, Y  +666.850, Z    +0.000, E1  +357.321, E3 -241989.510}
SPL {X  -159.990, Y  +662.495, Z    +0.000, E1  +351.318, E3 -241989.805}
SPL {X  -159.990, Y  +657.714, Z    +0.000, E1  +344.114, E3 -241990.366}
SPL {X  -159.990, Y  +651.822, Z    +0.000, E1  +335.261, E3 -241991.334}
SPL {X  -159.990, Y  +641.369, Z    +0.000, E1  +322.665, E3 -241994.172}
SPL {X  -159.990, Y  +598.251, Z    +0.000, E1  +304.104, E3 -242017.944}
SPL {X  -159.990, Y  +514.954, Z    +0.000, E1  +299.688, E3 -242091.739}
SPL {X  -159.990, Y  +505.641, Z    +0.000, E1  +299.707, E3 -242103.048}
SPL {X  -159.990, Y  +498.210, Z    +0.000, E1  +299.707, E3 -242112.042}
SPL {X  -159.990, Y  +488.988, Z    +0.000, E1  +299.693, E3 -242123.179}
SPL {X  -159.990, Y  +478.987, Z    +0.000, E1  +299.694, E3 -242135.281}
SPL {X  -159.990, Y  +468.796, Z    +0.000, E1  +299.698, E3 -242147.625}
SPL {X  -159.990, Y  +456.606, Z    +0.000, E1  +299.670, E3 -242162.331}
SPL {X  -159.990, Y  +443.890, Z    +0.000, E1  +299.691, E3 -242177.761}
SPL {X  -159.990, Y  +437.910, Z    +0.000, E1  +300.175, E3 -242188.232}
ENDSPLINE

SPLINE
SPL {X  -159.990, Y  +447.165, Z    +0.000, E1  +303.287, E3 -242196.787}
ENDSPLINE

SPLINE
SPL {X  -159.990, Y  +436.354, Z    +0.000, E1  +302.683, E3 -242207.798}
SPL {X  -159.990, Y  +425.140, Z    +0.000, E1  +301.982, E3 -242218.234}
SPL {X  -159.990, Y  +412.625, Z    +0.000, E1  +301.150, E3 -242229.070}
SPL {X  -159.990, Y  +398.951, Z    +0.000, E1  +300.353, E3 -242240.941}
SPL {X  -159.990, Y  +389.564, Z    +0.000, E1  +300.093, E3 -242250.755}
SPL {X  -159.985, Y  +381.230, Z    +0.000, E1  +300.090, E3 -242261.022}
SPL {X  -159.702, Y  +372.900, Z    +0.000, E1  +300.135, E3 -242271.559}
SPL {X  -159.030, Y  +365.001, Z    +0.000, E1  +300.230, E3 -242281.962}
SPL {X  -158.029, Y  +357.528, Z    +0.000, E1  +300.403, E3 -242292.217}
SPL {X  -156.953, Y  +351.476, Z    +0.000, E1  +300.570, E3 -242300.770}
SPL {X  -155.503, Y  +344.875, Z    +0.000, E1  +300.798, E3 -242310.380}
SPL {X  -153.622, Y  +337.813, Z    +0.000, E1  +301.097, E3 -242320.973}
SPL {X  -151.786, Y  +331.925, Z    +0.000, E1  +301.419, E3 -242330.094}
SPL {X  -150.141, Y  +327.233, Z    +0.000, E1  +301.695, E3 -242337.503}
SPL {X  -148.134, Y  +322.059, Z    +0.000, E1  +302.038, E3 -242345.837}
SPL {X  -145.832, Y  +316.699, Z    +0.000, E1  +302.442, E3 -242354.671}
SPL {X  -143.160, Y  +311.071, Z    +0.000, E1  +302.918, E3 -242364.116}
SPL {X  -140.427, Y  +305.839, Z    +0.000, E1  +303.430, E3 -242373.077}
SPL {X  -137.611, Y  +300.891, Z    +0.000, E1  +303.950, E3 -242381.654}
SPL {X  -121.335, Y  +278.219, Z    +0.000, E1  +311.699, E3 -242480.000}
ENDSPLINE

SPLINE
SPL {X  -146.770, Y  +318.818, Z    +0.000, E1  +325.496, E3 -242579.834}
SPL {X  -156.430, Y  +348.936, Z    +0.000, E1  +338.153, E3 -242596.565}
SPL {X  -159.088, Y  +365.539, Z    +0.000, E1  +347.196, E3 -242600.976}
SPL {X  -159.820, Y  +375.127, Z    +0.000, E1  +353.170, E3 -242602.399}
SPL {X  -159.990, Y  +382.134, Z    +0.000, E1  +357.935, E3 -242602.918}
SPL {X  -159.990, Y  +385.595, Z    +0.000, E1  +360.838, E3 -242603.033}
SPL {X  -159.990, Y  +390.176, Z    +0.000, E1  +366.367, E3 -242603.302}
SPL {X  -159.990, Y  +395.747, Z    +0.000, E1  +374.484, E3 -242603.927}
SPL {X  -159.990, Y  +402.387, Z    +0.000, E1  +384.140, E3 -242605.160}
SPL {X  -159.990, Y  +413.408, Z    +0.000, E1  +396.965, E3 -242608.461}
SPL {X  -159.990, Y  +455.723, Z    +0.000, E1  +415.803, E3 -242630.303}
SPL {X  -159.990, Y  +537.348, Z    +0.000, E1  +420.157, E3 -242702.896}
SPL {X  -159.990, Y  +545.972, Z    +0.000, E1  +420.143, E3 -242713.430}
SPL {X  -159.990, Y  +557.131, Z    +0.000, E1  +420.184, E3 -242726.944}
SPL {X  -159.990, Y  +569.073, Z    +0.000, E1  +420.153, E3 -242741.539}
SPL {X  -159.990, Y  +577.562, Z    +0.000, E1  +420.146, E3 -242751.879}
SPL {X  -159.990, Y  +585.415, Z    +0.000, E1  +420.147, E3 -242761.444}
SPL {X  -159.990, Y  +594.125, Z    +0.000, E1  +420.153, E3 -242772.030}
SPL {X  -159.990, Y  +602.716, Z    +0.000, E1  +420.150, E3 -242782.493}
SPL {X  -159.990, Y  +612.205, Z    +0.000, E1  +420.159, E3 -242794.030}
SPL {X  -159.990, Y  +624.752, Z    +0.000, E1  +420.194, E3 -242809.238}
SPL {X  -159.990, Y  +640.062, Z    +0.000, E1  +420.188, E3 -242827.901}
SPL {X  -159.990, Y  +652.098, Z    +0.000, E1  +420.153, E3 -242842.611}
SPL {X  -159.990, Y  +661.466, Z    +0.000, E1  +420.154, E3 -242854.022}
SPL {X  -159.963, Y  +674.441, Z    +0.000, E1  +420.189, E3 -242869.773}
SPL {X  -159.339, Y  +685.922, Z    +0.000, E1  +420.057, E3 -242884.452}
SPL {X  -158.381, Y  +694.132, Z    +0.000, E1  +419.909, E3 -242895.449}
SPL {X  -156.712, Y  +703.719, Z    +0.000, E1  +419.674, E3 -242908.814}
SPL {X  -154.922, Y  +711.450, Z    +0.000, E1  +419.348, E3 -242920.130}
SPL {X  -153.239, Y  +717.485, Z    +0.000, E1  +419.087, E3 -242929.162}
SPL {X  -150.608, Y  +725.483, Z    +0.000, E1  +418.677, E3 -242941.508}
SPL {X  -148.008, Y  +732.249, Z    +0.000, E1  +418.192, E3 -242952.374}
SPL {X  -145.943, Y  +737.055, Z    +0.000, E1  +417.829, E3 -242960.233}
SPL {X  -143.898, Y  +741.430, Z    +0.000, E1  +417.467, E3 -242967.502}
SPL {X  -141.624, Y  +745.927, Z    +0.000, E1  +417.045, E3 -242975.097}
SPL {X  -139.581, Y  +749.692, Z    +0.000, E1  +416.662, E3 -242981.544}
SPL {X  -137.120, Y  +753.931, Z    +0.000, E1  +416.213, E3 -242988.841}
SPL {X  -120.054, Y  +777.254, Z    +0.000, E1  +409.463, E3 -243075.587}
ENDSPLINE

SPLINE
SPL {X  -141.034, Y  +747.040, Z    +0.000, E1  +398.619, E3 -243183.749}
SPL {X  -152.334, Y  +720.400, Z    +0.000, E1  +389.143, E3 -243203.203}
SPL {X  -157.190, Y  +701.303, Z    +0.000, E1  +380.164, E3 -243210.364}
SPL {X  -159.460, Y  +684.516, Z    +0.000, E1  +370.556, E3 -243213.960}
SPL {X  -159.938, Y  +675.597, Z    +0.000, E1  +364.669, E3 -243214.966}
SPL {X  -159.990, Y  +671.043, Z    +0.000, E1  +361.371, E3 -243215.190}
SPL {X  -159.990, Y  +668.657, Z    +0.000, E1  +359.332, E3 -243215.250}
SPL {X  -159.990, Y  +665.812, Z    +0.000, E1  +355.875, E3 -243215.362}
SPL {X  -159.990, Y  +662.495, Z    +0.000, E1  +351.318, E3 -243215.611}
SPL {X  -159.990, Y  +657.714, Z    +0.000, E1  +344.114, E3 -243216.173}
SPL {X  -159.990, Y  +651.822, Z    +0.000, E1  +335.261, E3 -243217.141}
SPL {X  -159.990, Y  +641.369, Z    +0.000, E1  +322.665, E3 -243219.979}
SPL {X  -159.990, Y  +598.251, Z    +0.000, E1  +304.104, E3 -243243.750}
SPL {X  -159.990, Y  +514.954, Z    +0.000, E1  +299.688, E3 -243317.546}
SPL {X  -159.990, Y  +505.641, Z    +0.000, E1  +299.707, E3 -243328.855}
SPL {X  -159.990, Y  +498.210, Z    +0.000, E1  +299.707, E3 -243337.848}
SPL {X  -159.990, Y  +488.988, Z    +0.000, E1  +299.693, E3 -243348.985}
SPL {X  -159.990, Y  +478.987, Z    +0.000, E1  +299.694, E3 -243361.088}
SPL {X  -159.990, Y  +468.796, Z    +0.000, E1  +299.698, E3 -243373.432}
SPL {X  -159.990, Y  +456.606, Z    +0.000, E1  +299.670, E3 -243388.137}
SPL {X  -159.990, Y  +443.890, Z    +0.000, E1  +299.691, E3 -243403.567}
SPL {X  -159.990, Y  +437.910, Z    +0.000, E1  +300.175, E3 -243414.038}
ENDSPLINE

SPLINE
SPL {X  -159.990, Y  +447.165, Z    +0.000, E1  +303.287, E3 -243422.593}
ENDSPLINE

SPLINE
SPL {X  -159.990, Y  +436.354, Z    +0.000, E1  +302.683, E3 -243433.605}
SPL {X  -159.990, Y  +425.140, Z    +0.000, E1  +301.982, E3 -243444.040}
SPL {X  -159.990, Y  +412.625, Z    +0.000, E1  +301.150, E3 -243454.876}
SPL {X  -159.990, Y  +398.951, Z    +0.000, E1  +300.353, E3 -243466.747}
SPL {X  -159.990, Y  +389.564, Z    +0.000, E1  +300.093, E3 -243476.561}
SPL {X  -159.985, Y  +381.230, Z    +0.000, E1  +300.090, E3 -243486.828}
SPL {X  -159.702, Y  +372.900, Z    +0.000, E1  +300.135, E3 -243497.365}
SPL {X  -159.030, Y  +365.001, Z    +0.000, E1  +300.230, E3 -243507.768}
SPL {X  -158.029, Y  +357.528, Z    +0.000, E1  +300.403, E3 -243518.024}
SPL {X  -156.953, Y  +351.476, Z    +0.000, E1  +300.570, E3 -243526.577}
SPL {X  -155.503, Y  +344.875, Z    +0.000, E1  +300.798, E3 -243536.186}
SPL {X  -153.622, Y  +337.813, Z    +0.000, E1  +301.097, E3 -243546.780}
SPL {X  -150.877, Y  +329.275, Z    +0.000, E1  +301.527, E3 -243560.005}
SPL {X  -148.134, Y  +322.059, Z    +0.000, E1  +302.038, E3 -243571.643}
SPL {X  -145.832, Y  +316.699, Z    +0.000, E1  +302.442, E3 -243580.478}
SPL {X  -143.160, Y  +311.071, Z    +0.000, E1  +302.918, E3 -243589.923}
SPL {X  -139.570, Y  +304.288, Z    +0.000, E1  +303.552, E3 -243601.519}
SPL {X  -136.734, Y  +299.430, Z    +0.000, E1  +304.147, E3 -243610.057}
SPL {X  -121.335, Y  +278.219, Z    +0.000, E1  +311.699, E3 -243705.806}
ENDSPLINE

SPLINE
SPL {X  -146.770, Y  +318.818, Z    +0.000, E1  +325.496, E3 -243805.640}
SPL {X  -156.430, Y  +348.936, Z    +0.000, E1  +338.153, E3 -243822.371}
SPL {X  -159.088, Y  +365.539, Z    +0.000, E1  +347.196, E3 -243826.782}
SPL {X  -159.921, Y  +377.798, Z    +0.000, E1  +354.872, E3 -243828.442}
SPL {X  -159.990, Y  +383.148, Z    +0.000, E1  +358.786, E3 -243828.770}
SPL {X  -159.990, Y  +384.761, Z    +0.000, E1  +360.138, E3 -243828.814}
SPL {X  -159.990, Y  +387.385, Z    +0.000, E1  +362.811, E3 -243828.916}
SPL {X  -159.990, Y  +391.439, Z    +0.000, E1  +368.259, E3 -243829.213}
SPL {X  -159.990, Y  +395.747, Z    +0.000, E1  +374.484, E3 -243829.734}
SPL {X  -159.990, Y  +402.387, Z    +0.000, E1  +384.140, E3 -243830.966}
SPL {X  -159.990, Y  +414.244, Z    +0.000, E1  +397.704, E3 -243834.599}
SPL {X  -159.990, Y  +460.468, Z    +0.000, E1  +416.751, E3 -243858.691}
SPL {X  -159.990, Y  +537.348, Z    +0.000, E1  +420.157, E3 -243928.702}
SPL {X  -159.990, Y  +549.907, Z    +0.000, E1  +420.183, E3 -243943.960}
SPL {X  -159.990, Y  +560.677, Z    +0.000, E1  +420.145, E3 -243957.131}
SPL {X  -159.990, Y  +569.073, Z    +0.000, E1  +420.153, E3 -243967.345}
SPL {X  -159.990, Y  +581.828, Z    +0.000, E1  +420.191, E3 -243982.804}
SPL {X  -159.990, Y  +594.125, Z    +0.000, E1  +420.153, E3 -243997.837}
SPL {X  -159.990, Y  +602.716, Z    +0.000, E1  +420.150, E3 -244008.300}
SPL {X  -159.990, Y  +612.205, Z    +0.000, E1  +420.159, E3 -244019.836}
SPL {X  -159.990, Y  +620.604, Z    +0.000, E1  +420.153, E3 -244030.052}
SPL {X  -159.990, Y  +632.106, Z    +0.000, E1  +420.183, E3 -244044.028}
SPL {X  -159.990, Y  +643.341, Z    +0.000, E1  +420.148, E3 -244057.772}
SPL {X  -159.990, Y  +652.098, Z    +0.000, E1  +420.153, E3 -244068.417}
SPL {X  -159.990, Y  +661.466, Z    +0.000, E1  +420.154, E3 -244079.829}
SPL {X  -159.990, Y  +670.781, Z    +0.000, E1  +420.150, E3 -244091.176}
SPL {X  -159.839, Y  +678.445, Z    +0.000, E1  +420.123, E3 -244100.656}
SPL {X  -159.339, Y  +685.922, Z    +0.000, E1  +420.057, E3 -244110.258}
SPL {X  -158.381, Y  +694.132, Z    +0.000, E1  +419.909, E3 -244121.255}
SPL {X  -157.192, Y  +701.291, Z    +0.000, E1  +419.715, E3 -244131.226}
SPL {X  -155.426, Y  +709.440, Z    +0.000, E1  +419.459, E3 -244142.924}
SPL {X  -153.239, Y  +717.485, Z    +0.000, E1  +419.087, E3 -244154.969}
SPL {X  -151.467, Y  +723.022, Z    +0.000, E1  +418.780, E3 -244163.521}
SPL {X  -148.791, Y  +730.306, Z    +0.000, E1  +418.370, E3 -244174.986}
SPL {X  -145.943, Y  +737.055, Z    +0.000, E1  +417.829, E3 -244186.039}
SPL {X  -143.898, Y  +741.430, Z    +0.000, E1  +417.467, E3 -244193.308}
SPL {X  -140.579, Y  +747.882, Z    +0.000, E1  +416.895, E3 -244204.187}
SPL {X  -137.120, Y  +753.931, Z    +0.000, E1  +416.213, E3 -244214.648}
SPL {X  -120.054, Y  +777.254, Z    +0.000, E1  +409.463, E3 -244301.394}
ENDSPLINE

SPLINE
SPL {X  -141.034, Y  +747.040, Z    +0.000, E1  +398.619, E3 -244409.556}
SPL {X  -152.334, Y  +720.400, Z    +0.000, E1  +389.143, E3 -244429.010}
SPL {X  -157.190, Y  +701.303, Z    +0.000, E1  +380.164, E3 -244436.170}
SPL {X  -159.460, Y  +684.516, Z    +0.000, E1  +370.556, E3 -244439.766}
SPL {X  -159.938, Y  +675.597, Z    +0.000, E1  +364.669, E3 -244440.773}
SPL {X  -159.990, Y  +671.043, Z    +0.000, E1  +361.371, E3 -244440.996}
SPL {X  -159.990, Y  +668.657, Z    +0.000, E1  +359.332, E3 -244441.057}
SPL {X  -159.990, Y  +665.812, Z    +0.000, E1  +355.875, E3 -244441.168}
SPL {X  -159.990, Y  +662.495, Z    +0.000, E1  +351.318, E3 -244441.418}
SPL {X  -159.990, Y  +657.714, Z    +0.000, E1  +344.114, E3 -244441.979}
SPL {X  -159.990, Y  +651.822, Z    +0.000, E1  +335.261, E3 -244442.947}
SPL {X  -159.990, Y  +641.369, Z    +0.000, E1  +322.665, E3 -244445.785}
SPL {X  -159.990, Y  +598.251, Z    +0.000, E1  +304.104, E3 -244469.557}
SPL {X  -159.990, Y  +514.954, Z    +0.000, E1  +299.688, E3 -244543.352}
SPL {X  -159.990, Y  +505.641, Z    +0.000, E1  +299.707, E3 -244554.661}
SPL {X  -159.990, Y  +498.210, Z    +0.000, E1  +299.707, E3 -244563.655}
SPL {X  -159.990, Y  +488.988, Z    +0.000, E1  +299.693, E3 -244574.792}
SPL {X  -159.990, Y  +478.987, Z    +0.000, E1  +299.694, E3 -244586.894}
SPL {X  -159.990, Y  +468.796, Z    +0.000, E1  +299.698, E3 -244599.238}
SPL {X  -159.990, Y  +460.399, Z    +0.000, E1  +299.707, E3 -244609.415}
SPL {X  -159.990, Y  +453.289, Z    +0.000, E1  +299.707, E3 -244618.020}
SPL {X  -159.990, Y  +443.890, Z    +0.000, E1  +299.691, E3 -244629.374}
SPL {X  -159.990, Y  +437.910, Z    +0.000, E1  +300.175, E3 -244639.845}
ENDSPLINE

SPLINE
SPL {X  -159.990, Y  +447.165, Z    +0.000, E1  +303.287, E3 -244648.400}
ENDSPLINE

SPLINE
SPL {X  -159.990, Y  +436.354, Z    +0.000, E1  +302.683, E3 -244659.411}
SPL {X  -159.990, Y  +425.140, Z    +0.000, E1  +301.982, E3 -244669.847}
SPL {X  -159.990, Y  +412.625, Z    +0.000, E1  +301.150, E3 -244680.683}
SPL {X  -159.990, Y  +398.951, Z    +0.000, E1  +300.353, E3 -244692.554}
SPL {X  -159.990, Y  +389.564, Z    +0.000, E1  +300.093, E3 -244702.368}
SPL {X  -159.985, Y  +381.230, Z    +0.000, E1  +300.090, E3 -244712.635}
SPL {X  -159.702, Y  +372.900, Z    +0.000, E1  +300.135, E3 -244723.172}
SPL {X  -159.030, Y  +365.001, Z    +0.000, E1  +300.230, E3 -244733.575}
SPL {X  -158.029, Y  +357.528, Z    +0.000, E1  +300.403, E3 -244743.830}
SPL {X  -156.953, Y  +351.476, Z    +0.000, E1  +300.570, E3 -244752.383}
SPL {X  -155.503, Y  +344.875, Z    +0.000, E1  +300.798, E3 -244761.993}
SPL {X  -153.622, Y  +337.813, Z    +0.000, E1  +301.097, E3 -244772.586}
SPL {X  -150.877, Y  +329.275, Z    +0.000, E1  +301.527, E3 -244785.811}
SPL {X  -148.134, Y  +322.059, Z    +0.000, E1  +302.038, E3 -244797.450}
SPL {X  -145.832, Y  +316.699, Z    +0.000, E1  +302.442, E3 -244806.284}
SPL {X  -143.160, Y  +311.071, Z    +0.000, E1  +302.918, E3 -244815.729}
SPL {X  -140.427, Y  +305.839, Z    +0.000, E1  +303.430, E3 -244824.690}
SPL {X  -137.611, Y  +300.891, Z    +0.000, E1  +303.950, E3 -244833.266}
SPL {X  -121.335, Y  +278.219, Z    +0.000, E1  +311.699, E3 -244931.613}
ENDSPLINE

SPLINE
SPL {X  -146.770, Y  +318.818, Z    +0.000, E1  +325.496, E3 -245031.446}
SPL {X  -156.430, Y  +348.936, Z    +0.000, E1  +338.153, E3 -245048.178}
SPL {X  -159.088, Y  +365.539, Z    +0.000, E1  +347.196, E3 -245052.589}
SPL {X  -159.921, Y  +377.798, Z    +0.000, E1  +354.872, E3 -245054.249}
SPL {X  -159.990, Y  +384.169, Z    +0.000, E1  +359.534, E3 -245054.604}
SPL {X  -159.990, Y  +387.385, Z    +0.000, E1  +362.811, E3 -245054.723}
SPL {X  -159.990, Y  +391.439, Z    +0.000, E1  +368.259, E3 -245055.019}
SPL {X  -159.990, Y  +395.747, Z    +0.000, E1  +374.484, E3 -245055.540}
SPL {X  -159.990, Y  +402.387, Z    +0.000, E1  +384.140, E3 -245056.772}
SPL {X  -159.990, Y  +414.244, Z    +0.000, E1  +397.704, E3 -245060.405}
SPL {X  -159.990, Y  +460.468, Z    +0.000, E1  +416.751, E3 -245084.497}
SPL {X  -159.990, Y  +537.348, Z    +0.000, E1  +420.157, E3 -245154.509}
SPL {X  -159.990, Y  +549.907, Z    +0.000, E1  +420.183, E3 -245169.766}
SPL {X  -159.990, Y  +560.677, Z    +0.000, E1  +420.145, E3 -245182.937}
SPL {X  -159.990, Y  +569.073, Z    +0.000, E1  +420.153, E3 -245193.152}
SPL {X  -159.990, Y  +581.828, Z    +0.000, E1  +420.191, E3 -245208.611}
SPL {X  -159.990, Y  +594.125, Z    +0.000, E1  +420.153, E3 -245223.643}
SPL {X  -159.990, Y  +602.716, Z    +0.000, E1  +420.150, E3 -245234.106}
SPL {X  -159.990, Y  +612.205, Z    +0.000, E1  +420.159, E3 -245245.643}
SPL {X  -159.990, Y  +620.604, Z    +0.000, E1  +420.153, E3 -245255.858}
SPL {X  -159.990, Y  +632.106, Z    +0.000, E1  +420.183, E3 -245269.835}
SPL {X  -159.990, Y  +643.341, Z    +0.000, E1  +420.148, E3 -245283.578}
SPL {X  -159.990, Y  +652.098, Z    +0.000, E1  +420.153, E3 -245294.224}
SPL {X  -159.990, Y  +661.466, Z    +0.000, E1  +420.154, E3 -245305.635}
SPL {X  -159.990, Y  +670.781, Z    +0.000, E1  +420.150, E3 -245316.983}
SPL {X  -159.839, Y  +678.445, Z    +0.000, E1  +420.123, E3 -245326.462}
SPL {X  -159.339, Y  +685.922, Z    +0.000, E1  +420.057, E3 -245336.065}
SPL {X  -158.381, Y  +694.132, Z    +0.000, E1  +419.909, E3 -245347.062}
SPL {X  -157.192, Y  +701.291, Z    +0.000, E1  +419.715, E3 -245357.032}
SPL {X  -155.426, Y  +709.440, Z    +0.000, E1  +419.459, E3 -245368.730}
SPL {X  -153.239, Y  +717.485, Z    +0.000, E1  +419.087, E3 -245380.775}
SPL {X  -150.608, Y  +725.483, Z    +0.000, E1  +418.677, E3 -245393.120}
SPL {X  -148.008, Y  +732.249, Z    +0.000, E1  +418.192, E3 -245403.987}
SPL {X  -145.943, Y  +737.055, Z    +0.000, E1  +417.829, E3 -245411.846}
SPL {X  -143.898, Y  +741.430, Z    +0.000, E1  +417.467, E3 -245419.115}
SPL {X  -140.579, Y  +747.882, Z    +0.000, E1  +416.895, E3 -245429.994}
SPL {X  -137.120, Y  +753.931, Z    +0.000, E1  +416.213, E3 -245440.454}
SPL {X  -120.054, Y  +777.254, Z    +0.000, E1  +409.463, E3 -245527.200}
ENDSPLINE

SPLINE
SPL {X  -141.034, Y  +747.040, Z    +0.000, E1  +398.619, E3 -245635.362}
SPL {X  -152.334, Y  +720.400, Z    +0.000, E1  +389.143, E3 -245654.816}
SPL {X  -157.190, Y  +701.303, Z    +0.000, E1  +380.164, E3 -245661.977}
SPL {X  -159.460, Y  +684.516, Z    +0.000, E1  +370.556, E3 -245665.572}
SPL {X  -159.938, Y  +675.597, Z    +0.000, E1  +364.669, E3 -245666.579}
SPL {X  -159.990, Y  +669.975, Z    +0.000, E1  +360.595, E3 -245666.829}
SPL {X  -159.990, Y  +666.850, Z    +0.000, E1  +357.321, E3 -245666.930}
SPL {X  -159.990, Y  +662.495, Z    +0.000, E1  +351.318, E3 -245667.224}
SPL {X  -159.990, Y  +657.714, Z    +0.000, E1  +344.114, E3 -245667.785}
SPL {X  -159.990, Y  +651.822, Z    +0.000, E1  +335.261, E3 -245668.754}
SPL {X  -159.990, Y  +641.369, Z    +0.000, E1  +322.665, E3 -245671.592}
SPL {X  -159.990, Y  +598.251, Z    +0.000, E1  +304.104, E3 -245695.363}
SPL {X  -159.990, Y  +514.954, Z    +0.000, E1  +299.688, E3 -245769.159}
SPL {X  -159.990, Y  +501.679, Z    +0.000, E1  +299.667, E3 -245785.196}
SPL {X  -159.990, Y  +488.988, Z    +0.000, E1  +299.693, E3 -245800.598}
SPL {X  -159.990, Y  +478.987, Z    +0.000, E1  +299.694, E3 -245812.701}
SPL {X  -159.990, Y  +468.796, Z    +0.000, E1  +299.698, E3 -245825.044}
SPL {X  -159.990, Y  +460.399, Z    +0.000, E1  +299.707, E3 -245835.221}
SPL {X  -159.990, Y  +453.289, Z    +0.000, E1  +299.707, E3 -245843.827}
SPL {X  -159.990, Y  +443.890, Z    +0.000, E1  +299.691, E3 -245855.180}
SPL {X  -159.990, Y  +437.910, Z    +0.000, E1  +300.175, E3 -245865.651}
ENDSPLINE

SPLINE
SPL {X  -159.990, Y  +447.165, Z    +0.000, E1  +303.287, E3 -245874.206}
ENDSPLINE

SPLINE
SPL {X  -159.990, Y  +436.354, Z    +0.000, E1  +302.683, E3 -245885.218}
SPL {X  -159.990, Y  +425.140, Z    +0.000, E1  +301.982, E3 -245895.653}
SPL {X  -159.990, Y  +412.625, Z    +0.000, E1  +301.150, E3 -245906.489}
SPL {X  -159.990, Y  +398.951, Z    +0.000, E1  +300.353, E3 -245918.360}
SPL {X  -159.990, Y  +389.564, Z    +0.000, E1  +300.093, E3 -245928.174}
SPL {X  -159.985, Y  +381.230, Z    +0.000, E1  +300.090, E3 -245938.441}
SPL {X  -159.702, Y  +372.900, Z    +0.000, E1  +300.135, E3 -245948.978}
SPL {X  -159.030, Y  +365.001, Z    +0.000, E1  +300.230, E3 -245959.381}
SPL {X  -157.449, Y  +354.098, Z    +0.000, E1  +300.447, E3 -245974.381}
SPL {X  -155.503, Y  +344.875, Z    +0.000, E1  +300.798, E3 -245987.799}
SPL {X  -153.622, Y  +337.813, Z    +0.000, E1  +301.097, E3 -245998.393}
SPL {X  -150.877, Y  +329.275, Z    +0.000, E1  +301.527, E3 -246011.618}
SPL {X  -148.134, Y  +322.059, Z    +0.000, E1  +302.038, E3 -246023.256}
SPL {X  -145.832, Y  +316.699, Z    +0.000, E1  +302.442, E3 -246032.090}
SPL {X  -143.160, Y  +311.071, Z    +0.000, E1  +302.918, E3 -246041.536}
SPL {X  -140.427, Y  +305.839, Z    +0.000, E1  +303.430, E3 -246050.497}
SPL {X  -137.611, Y  +300.891, Z    +0.000, E1  +303.950, E3 -246059.073}
SPL {X  -121.335, Y  +278.219, Z    +0.000, E1  +311.699, E3 -246157.419}
ENDSPLINE

SPLINE
SPL {X  -146.770, Y  +318.818, Z    +0.000, E1  +325.496, E3 -246257.253}
SPL {X  -156.430, Y  +348.936, Z    +0.000, E1  +338.153, E3 -246273.984}
SPL {X  -159.088, Y  +365.539, Z    +0.000, E1  +347.196, E3 -246278.395}
SPL {X  -159.921, Y  +377.798, Z    +0.000, E1  +354.872, E3 -246280.055}
SPL {X  -159.990, Y  +383.148, Z    +0.000, E1  +358.786, E3 -246280.383}
SPL {X  -159.990, Y  +385.595, Z    +0.000, E1  +360.838, E3 -246280.452}
SPL {X  -159.990, Y  +390.176, Z    +0.000, E1  +366.367, E3 -246280.721}
SPL {X  -159.990, Y  +395.747, Z    +0.000, E1  +374.484, E3 -246281.346}
SPL {X  -159.990, Y  +402.387, Z    +0.000, E1  +384.140, E3 -246282.579}
SPL {X  -159.990, Y  +413.408, Z    +0.000, E1  +396.965, E3 -246285.880}
SPL {X  -159.990, Y  +455.723, Z    +0.000, E1  +415.803, E3 -246307.723}
SPL {X  -159.990, Y  +537.348, Z    +0.000, E1  +420.157, E3 -246380.315}
SPL {X  -159.990, Y  +549.907, Z    +0.000, E1  +420.183, E3 -246395.573}
SPL {X  -159.990, Y  +560.677, Z    +0.000, E1  +420.145, E3 -246408.744}
SPL {X  -159.990, Y  +569.073, Z    +0.000, E1  +420.153, E3 -246418.958}
SPL {X  -159.990, Y  +581.828, Z    +0.000, E1  +420.191, E3 -246434.417}
SPL {X  -159.990, Y  +594.125, Z    +0.000, E1  +420.153, E3 -246449.450}
SPL {X  -159.990, Y  +602.716, Z    +0.000, E1  +420.150, E3 -246459.913}
SPL {X  -159.990, Y  +612.205, Z    +0.000, E1  +420.159, E3 -246471.449}
SPL {X  -159.990, Y  +620.604, Z    +0.000, E1  +420.153, E3 -246481.665}
SPL {X  -159.990, Y  +632.106, Z    +0.000, E1  +420.183, E3 -246495.641}
SPL {X  -159.990, Y  +643.341, Z    +0.000, E1  +420.148, E3 -246509.385}
SPL {X  -159.990, Y  +652.098, Z    +0.000, E1  +420.153, E3 -246520.030}
SPL {X  -159.990, Y  +661.466, Z    +0.000, E1  +420.154, E3 -246531.441}
SPL {X  -159.963, Y  +674.441, Z    +0.000, E1  +420.189, E3 -246547.192}
SPL {X  -159.339, Y  +685.922, Z    +0.000, E1  +420.057, E3 -246561.871}
SPL {X  -158.381, Y  +694.132, Z    +0.000, E1  +419.909, E3 -246572.868}
SPL {X  -156.712, Y  +703.719, Z    +0.000, E1  +419.674, E3 -246586.233}
SPL {X  -154.922, Y  +711.450, Z    +0.000, E1  +419.348, E3 -246597.549}
SPL {X  -153.239, Y  +717.485, Z    +0.000, E1  +419.087, E3 -246606.582}
SPL {X  -150.608, Y  +725.483, Z    +0.000, E1  +418.677, E3 -246618.927}
SPL {X  -148.008, Y  +732.249, Z    +0.000, E1  +418.192, E3 -246629.793}
SPL {X  -145.943, Y  +737.055, Z    +0.000, E1  +417.829, E3 -246637.652}
SPL {X  -143.898, Y  +741.430, Z    +0.000, E1  +417.467, E3 -246644.921}
SPL {X  -141.624, Y  +745.927, Z    +0.000, E1  +417.045, E3 -246652.517}
SPL {X  -139.581, Y  +749.692, Z    +0.000, E1  +416.662, E3 -246658.963}
SPL {X  -137.120, Y  +753.931, Z    +0.000, E1  +416.213, E3 -246666.261}
SPL {X  -120.054, Y  +777.254, Z    +0.000, E1  +409.463, E3 -246753.007}
ENDSPLINE

SPLINE
SPL {X  -141.034, Y  +747.040, Z    +0.000, E1  +398.619, E3 -246861.168}
SPL {X  -152.334, Y  +720.400, Z    +0.000, E1  +389.143, E3 -246880.623}
SPL {X  -157.190, Y  +701.303, Z    +0.000, E1  +380.164, E3 -246887.783}
SPL {X  -159.460, Y  +684.516, Z    +0.000, E1  +370.556, E3 -246891.379}
SPL {X  -159.938, Y  +675.597, Z    +0.000, E1  +364.669, E3 -246892.385}
SPL {X  -159.990, Y  +669.975, Z    +0.000, E1  +360.595, E3 -246892.636}
SPL {X  -159.990, Y  +666.850, Z    +0.000, E1  +357.321, E3 -246892.736}
SPL {X  -159.990, Y  +662.495, Z    +0.000, E1  +351.318, E3 -246893.031}
SPL {X  -159.990, Y  +657.714, Z    +0.000, E1  +344.114, E3 -246893.592}
SPL {X  -159.990, Y  +651.822, Z    +0.000, E1  +335.261, E3 -246894.560}
SPL {X  -159.990, Y  +641.369, Z    +0.000, E1  +322.665, E3 -246897.398}
SPL {X  -159.990, Y  +598.251, Z    +0.000, E1  +304.104, E3 -246921.170}
SPL {X  -159.990, Y  +514.954, Z    +0.000, E1  +299.688, E3 -246994.965}
SPL {X  -159.990, Y  +505.641, Z    +0.000, E1  +299.707, E3 -247006.274}
SPL {X  -159.990, Y  +498.210, Z    +0.000, E1  +299.707, E3 -247015.268}
SPL {X  -159.990, Y  +488.988, Z    +0.000, E1  +299.693, E3 -247026.404}
SPL {X  -159.990, Y  +478.987, Z    +0.000, E1  +299.694, E3 -247038.507}
SPL {X  -159.990, Y  +468.796, Z    +0.000, E1  +299.698, E3 -247050.851}
SPL {X  -159.990, Y  +460.399, Z    +0.000, E1  +299.707, E3 -247061.028}
SPL {X  -159.990, Y  +453.289, Z    +0.000, E1  +299.707, E3 -247069.633}
SPL {X  -159.990, Y  +443.890, Z    +0.000, E1  +299.691, E3 -247080.987}
SPL {X  -159.990, Y  +437.910, Z    +0.000, E1  +300.175, E3 -247091.458}
ENDSPLINE

SPLINE
SPL {X  -159.990, Y  +447.165, Z    +0.000, E1  +303.287, E3 -247100.013}
ENDSPLINE

SPLINE
SPL {X  -159.990, Y  +436.354, Z    +0.000, E1  +302.683, E3 -247111.024}
SPL {X  -159.990, Y  +425.140, Z    +0.000, E1  +301.982, E3 -247121.459}
SPL {X  -159.990, Y  +412.625, Z    +0.000, E1  +301.150, E3 -247132.296}
SPL {X  -159.990, Y  +398.951, Z    +0.000, E1  +300.353, E3 -247144.167}
SPL {X  -159.990, Y  +389.564, Z    +0.000, E1  +300.093, E3 -247153.981}
SPL {X  -159.985, Y  +381.230, Z    +0.000, E1  +300.090, E3 -247164.248}
SPL {X  -159.702, Y  +372.900, Z    +0.000, E1  +300.135, E3 -247174.785}
SPL {X  -159.030, Y  +365.001, Z    +0.000, E1  +300.230, E3 -247185.188}
SPL {X  -157.449, Y  +354.098, Z    +0.000, E1  +300.447, E3 -247200.187}
SPL {X  -155.503, Y  +344.875, Z    +0.000, E1  +300.798, E3 -247213.606}
SPL {X  -153.622, Y  +337.813, Z    +0.000, E1  +301.097, E3 -247224.199}
SPL {X  -150.877, Y  +329.275, Z    +0.000, E1  +301.527, E3 -247237.424}
SPL {X  -148.134, Y  +322.059, Z    +0.000, E1  +302.038, E3 -247249.063}
SPL {X  -145.832, Y  +316.699, Z    +0.000, E1  +302.442, E3 -247257.897}
SPL {X  -143.160, Y  +311.071, Z    +0.000, E1  +302.918, E3 -247267.342}
SPL {X  -140.427, Y  +305.839, Z    +0.000, E1  +303.430, E3 -247276.303}
SPL {X  -137.611, Y  +300.891, Z    +0.000, E1  +303.950, E3 -247284.879}
SPL {X  -121.335, Y  +278.219, Z    +0.000, E1  +311.699, E3 -247383.225}
ENDSPLINE

